LIN {X 0,Y 571.176,Z 836.782,A -85,B 0,C 180,E1 -9234.219,E2 -9234.219} C_VEL
LIN {X 0,Y 568.338,Z 859.351,A -85,B 0,C 180,E1 -9235.423,E2 -9235.423} C_VEL
LIN {X 0,Y 565.653,Z 878.944,A -85,B 0,C 180,E1 -9236.651,E2 -9236.651} C_VEL
LIN {X 0,Y 562.465,Z 900.787,A -85,B 0,C 180,E1 -9238.251,E2 -9238.251} C_VEL
LIN {X 0,Y 559.839,Z 917.889,A -85,B 0,C 180,E1 -9239.698,E2 -9239.698} C_VEL
LIN {X 0,Y 556.887,Z 936.762,A -85,B 0,C 180,E1 -9241.522,E2 -9241.522} C_VEL
LIN {X 0,Y 554.378,Z 952.803,A -85,B 0,C 180,E1 -9243.314,E2 -9243.314} C_VEL
LIN {X 0,Y 551.914,Z 969.075,A -85,B 0,C 180,E1 -9245.375,E2 -9245.375} C_VEL
LIN {X 0,Y 549.794,Z 983.496,A -85,B 0,C 180,E1 -9247.501,E2 -9247.501} C_VEL
LIN {X 0,Y 548.027,Z 996.716,A -85,B 0,C 180,E1 -9249.717,E2 -9249.717} C_VEL
LIN {X 0,Y 546.569,Z 1008.744,A -85,B 0,C 180,E1 -9252.101,E2 -9252.101} C_VEL
LIN {X 0,Y 545.53,Z 1019.1,A -85,B 0,C 180,E1 -9254.479,E2 -9254.479} C_VEL
LIN {X 0,Y 544.771,Z 1027.944,A -85,B 0,C 180,E1 -9256.953,E2 -9256.953} C_VEL
LIN {X 0,Y 544.345,Z 1034.638,A -85,B 0,C 180,E1 -9259.201,E2 -9259.201} C_VEL
LIN {X 0,Y 544.06,Z 1040.823,A -85,B 0,C 180,E1 -9261.865,E2 -9261.865} C_VEL
LIN {X 0,Y 543.971,Z 1044.474,A -85,B 0,C 180,E1 -9263.986,E2 -9263.986} C_VEL
LIN {X 0,Y 543.924,Z 1047.387,A -85,B 0,C 180,E1 -9266.417,E2 -9266.417} C_VEL
LIN {X 0,Y 543.915,Z 1048.764,A -85,B 0,C 180,E1 -9268.947,E2 -9268.947} C_VEL
LIN {X 0,Y 543.919,Z 1048.761,A -85,B 0,C 180,E1 -9271.159,E2 -9271.159} C_VEL
LIN {X 0,Y 543.927,Z 1047.259,A -85,B 0,C 180,E1 -9273.795,E2 -9273.795} C_VEL
LIN {X 0,Y 543.971,Z 1044.452,A -85,B 0,C 180,E1 -9276.12,E2 -9276.12} C_VEL
LIN {X 0,Y 544.08,Z 1040.589,A -85,B 0,C 180,E1 -9278.348,E2 -9278.348} C_VEL
LIN {X 0,Y 544.362,Z 1034.293,A -85,B 0,C 180,E1 -9281.013,E2 -9281.013} C_VEL
LIN {X 0,Y 544.777,Z 1027.888,A -85,B 0,C 180,E1 -9283.155,E2 -9283.155} C_VEL
LIN {X 0,Y 545.538,Z 1019.019,A -85,B 0,C 180,E1 -9285.63,E2 -9285.63} C_VEL
LIN {X 0,Y 546.583,Z 1008.645,A -85,B 0,C 180,E1 -9288.009,E2 -9288.009} C_VEL
LIN {X 0,Y 548.043,Z 996.594,A -85,B 0,C 180,E1 -9290.394,E2 -9290.394} C_VEL
LIN {X 0,Y 549.866,Z 982.95,A -85,B 0,C 180,E1 -9292.675,E2 -9292.675} C_VEL
LIN {X 0,Y 552.067,Z 968.089,A -85,B 0,C 180,E1 -9294.851,E2 -9294.851} C_VEL
LIN {X 0,Y 554.409,Z 952.604,A -85,B 0,C 180,E1 -9296.8,E2 -9296.8} C_VEL
LIN {X 0,Y 557.001,Z 936.1,A -85,B 0,C 180,E1 -9298.64,E2 -9298.64} C_VEL
LIN {X 0,Y 559.829,Z 918.013,A -85,B 0,C 180,E1 -9300.382,E2 -9300.382} C_VEL
LIN {X 0,Y 562.409,Z 901.202,A -85,B 0,C 180,E1 -9301.807,E2 -9301.807} C_VEL
LIN {X 0,Y 565.502,Z 880.175,A -85,B 0,C 180,E1 -9303.36,E2 -9303.36} C_VEL
LIN {X 0,Y 568.145,Z 860.831,A -85,B 0,C 180,E1 -9304.581,E2 -9304.581} C_VEL
LIN {X 0,Y 570.995,Z 838.465,A -85,B 0,C 180,E1 -9305.795,E2 -9305.795} C_VEL
LIN {X 0,Y 573.356,Z 817.368,A -85,B 0,C 180,E1 -9306.739,E2 -9306.739} C_VEL
LIN {X 0,Y 575.397,Z 796.537,A -85,B 0,C 180,E1 -9307.523,E2 -9307.523} C_VEL
LIN {X 0,Y 577.39,Z 771.878,A -85,B 0,C 180,E1 -9308.254,E2 -9308.254} C_VEL
LIN {X 0,Y 578.666,Z 751.524,A -85,B 0,C 180,E1 -9308.716,E2 -9308.716} C_VEL
LIN {X 0,Y 579.729,Z 725.617,A -85,B 0,C 180,E1 -9309.143,E2 -9309.143} C_VEL
LIN {X 0,Y 586.415,Z 471.71,A -85,B 0,C 180,E1 -9312.634,E2 -9312.634} C_VEL
LIN {X 0,Y 587.803,Z 417.401,A -85,B 0,C 180,E1 -9313.399,E2 -9313.399} C_VEL
LIN {X 0,Y 574.092,Z 395,A -85,B 0,C 180,E1 -9315.104,E2 -9315.104} C_VEL
LIN {X 0,Y 562.129,Z 377.006,A -85,B 0,C 180,E1 -9316.677,E2 -9316.677} C_VEL
LIN {X 0,Y 555.49,Z 368.058,A -85,B 0,C 180,E1 -9317.58,E2 -9317.58} C_VEL
LIN {X 0,Y 552.526,Z 363.838,A -85,B 0,C 180,E1 -9318,E2 -9318} C_VEL
LIN {X 0,Y 549.725,Z 359.959,A -85,B 0,C 180,E1 -9318.402,E2 -9318.402} C_VEL
LIN {X 0,Y 548.841,Z 358.788,A -85,B 0,C 180,E1 -9318.529,E2 -9318.529} C_VEL
LIN {X 0,Y 546.385,Z 356.008,A -85,B 0,C 180,E1 -9318.878,E2 -9318.878} C_VEL
LIN {X 0,Y 545.511,Z 353.224,A -85,B 0,C 180,E1 -9319.041,E2 -9319.041} C_VEL
LIN {X 0,Y 545.509,Z 353.268,A -85,B 0,C 180,E1 -9322.383,E2 -9322.383} C_VEL
LIN {X 0,Y 545.559,Z 353.26,A -85,B 0,C 180,E1 -9325.632,E2 -9325.632} C_VEL
LIN {X 0,Y 545.501,Z 353.265,A -85,B 0,C 180,E1 -9328.875,E2 -9328.875} C_VEL
LIN {X 0,Y 545.543,Z 353.258,A -85,B 0,C 180,E1 -9332.136,E2 -9332.136} C_VEL
LIN {X 0,Y 545.515,Z 353.271,A -85,B 0,C 180,E1 -9335.297,E2 -9335.297} C_VEL
LIN {X 0,Y 545.507,Z 353.277,A -85,B 0,C 180,E1 -9338.72,E2 -9338.72} C_VEL
LIN {X 0,Y 545.562,Z 353.271,A -85,B 0,C 180,E1 -9341.956,E2 -9341.956} C_VEL
LIN {X 0,Y 545.5,Z 353.262,A -85,B 0,C 180,E1 -9345.239,E2 -9345.239} C_VEL
LIN {X 0,Y 545.524,Z 353.257,A -85,B 0,C 180,E1 -9348.583,E2 -9348.583} C_VEL
LIN {X 0,Y 545.533,Z 353.279,A -85,B 0,C 180,E1 -9351.79,E2 -9351.79} C_VEL
LIN {X 0,Y 545.502,Z 353.273,A -85,B 0,C 180,E1 -9355.058,E2 -9355.058} C_VEL
LIN {X 0,Y 545.562,Z 353.252,A -85,B 0,C 180,E1 -9358.32,E2 -9358.32} C_VEL
LIN {X 0,Y 545.501,Z 353.279,A -85,B 0,C 180,E1 -9361.47,E2 -9361.47} C_VEL
LIN {X 0,Y 545.528,Z 353.276,A -85,B 0,C 180,E1 -9364.837,E2 -9364.837} C_VEL
LIN {X 0,Y 545.525,Z 353.257,A -85,B 0,C 180,E1 -9368.007,E2 -9368.007} C_VEL
LIN {X 0,Y 545.503,Z 353.271,A -85,B 0,C 180,E1 -9371.311,E2 -9371.311} C_VEL
LIN {X 0,Y 545.571,Z 353.272,A -85,B 0,C 180,E1 -9374.605,E2 -9374.605} C_VEL
LIN {X 0,Y 545.503,Z 353.27,A -85,B 0,C 180,E1 -9377.825,E2 -9377.825} C_VEL
LIN {X 0,Y 545.522,Z 353.261,A -85,B 0,C 180,E1 -9381.167,E2 -9381.167} C_VEL
LIN {X 0,Y 545.522,Z 353.262,A -85,B 0,C 180,E1 -9384.241,E2 -9384.241} C_VEL
LIN {X 0,Y 545.503,Z 353.267,A -85,B 0,C 180,E1 -9387.629,E2 -9387.629} C_VEL
LIN {X 0,Y 545.571,Z 353.262,A -85,B 0,C 180,E1 -9390.753,E2 -9390.753} C_VEL
LIN {X 0,Y 545.502,Z 353.27,A -85,B 0,C 180,E1 -9394.055,E2 -9394.055} C_VEL
LIN {X 0,Y 545.53,Z 353.267,A -85,B 0,C 180,E1 -9397.35,E2 -9397.35} C_VEL
LIN {X 0,Y 545.578,Z 353.397,A -85,B 0,C 180,E1 -9398.84,E2 -9398.84} C_VEL
LIN {X 0,Y 546.798,Z 356.681,A -85,B 0,C 180,E1 -9399.386,E2 -9399.386} C_VEL
LIN {X 0,Y 552.392,Z 369.121,A -85,B 0,C 180,E1 -9401.491,E2 -9401.491} C_VEL
LIN {X 0,Y 553.905,Z 372.53,A -85,B 0,C 180,E1 -9401.993,E2 -9401.993} C_VEL
LIN {X 0,Y 567.117,Z 392.673,A -85,B 0,C 180,E1 -9403.808,E2 -9403.808} C_VEL
LIN {X 0,Y 577.736,Z 409.877,A -85,B 0,C 180,E1 -9405.184,E2 -9405.184} C_VEL
LIN {X 0,Y 587.88,Z 427.42,A -85,B 0,C 180,E1 -9406.442,E2 -9406.442} C_VEL
LIN {X 0,Y 580.977,Z 687.347,A -85,B 0,C 180,E1 -9410.026,E2 -9410.026} C_VEL
LIN {X 0,Y 578.837,Z 765.694,A -85,B 0,C 180,E1 -9411.119,E2 -9411.119} C_VEL
LIN {X 0,Y 577.261,Z 791.324,A -85,B 0,C 180,E1 -9411.637,E2 -9411.637} C_VEL
LIN {X 0,Y 575.512,Z 813.307,A -85,B 0,C 180,E1 -9412.236,E2 -9412.236} C_VEL
LIN {X 0,Y 573.112,Z 838.377,A -85,B 0,C 180,E1 -9413.118,E2 -9413.118} C_VEL
LIN {X 0,Y 570.954,Z 857.811,A -85,B 0,C 180,E1 -9413.955,E2 -9413.955} C_VEL
LIN {X 0,Y 568.235,Z 880.101,A -85,B 0,C 180,E1 -9415.085,E2 -9415.085} C_VEL
LIN {X 0,Y 565.429,Z 900.717,A -85,B 0,C 180,E1 -9416.334,E2 -9416.334} C_VEL
LIN {X 0,Y 562.638,Z 920.354,A -85,B 0,C 180,E1 -9417.699,E2 -9417.699} C_VEL
LIN {X 0,Y 559.633,Z 940.46,A -85,B 0,C 180,E1 -9419.329,E2 -9419.329} C_VEL
LIN {X 0,Y 557.091,Z 957.393,A -85,B 0,C 180,E1 -9420.896,E2 -9420.896} C_VEL
LIN {X 0,Y 554.163,Z 976.778,A -85,B 0,C 180,E1 -9422.955,E2 -9422.955} C_VEL
LIN {X 0,Y 551.957,Z 991.957,A -85,B 0,C 180,E1 -9424.804,E2 -9424.804} C_VEL
LIN {X 0,Y 549.688,Z 1008.329,A -85,B 0,C 180,E1 -9427.091,E2 -9427.091} C_VEL
LIN {X 0,Y 548.053,Z 1021.183,A -85,B 0,C 180,E1 -9429.16,E2 -9429.16} C_VEL
LIN {X 0,Y 546.495,Z 1034.957,A -85,B 0,C 180,E1 -9431.73,E2 -9431.73} C_VEL
LIN {X 0,Y 545.565,Z 1044.545,A -85,B 0,C 180,E1 -9433.824,E2 -9433.824} C_VEL
LIN {X 0,Y 544.805,Z 1054.264,A -85,B 0,C 180,E1 -9436.305,E2 -9436.305} C_VEL
LIN {X 0,Y 544.339,Z 1061.766,A -85,B 0,C 180,E1 -9438.665,E2 -9438.665} C_VEL
LIN {X 0,Y 544.07,Z 1067.86,A -85,B 0,C 180,E1 -9441.013,E2 -9441.013} C_VEL
LIN {X 0,Y 543.949,Z 1072.768,A -85,B 0,C 180,E1 -9443.562,E2 -9443.562} C_VEL
LIN {X 0,Y 543.918,Z 1075.605,A -85,B 0,C 180,E1 -9445.677,E2 -9445.677} C_VEL
LIN {X 0,Y 543.91,Z 1077.486,A -85,B 0,C 180,E1 -9447.998,E2 -9447.998} C_VEL
LIN {X 0,Y 543.902,Z 1077.918,A -85,B 0,C 180,E1 -9450.527,E2 -9450.527} C_VEL
LIN {X 0,Y 543.912,Z 1077.002,A -85,B 0,C 180,E1 -9452.739,E2 -9452.739} C_VEL
LIN {X 0,Y 543.933,Z 1074.678,A -85,B 0,C 180,E1 -9455.168,E2 -9455.168} C_VEL
LIN {X 0,Y 543.986,Z 1070.708,A -85,B 0,C 180,E1 -9457.605,E2 -9457.605} C_VEL
LIN {X 0,Y 544.145,Z 1066.052,A -85,B 0,C 180,E1 -9459.733,E2 -9459.733} C_VEL
LIN {X 0,Y 544.483,Z 1059.283,A -85,B 0,C 180,E1 -9462.192,E2 -9462.192} C_VEL
LIN {X 0,Y 545.03,Z 1051.049,A -85,B 0,C 180,E1 -9464.556,E2 -9464.556} C_VEL
LIN {X 0,Y 545.787,Z 1042.224,A -85,B 0,C 180,E1 -9466.716,E2 -9466.716} C_VEL
LIN {X 0,Y 547.006,Z 1030.198,A -85,B 0,C 180,E1 -9469.21,E2 -9469.21} C_VEL
LIN {X 0,Y 548.367,Z 1018.538,A -85,B 0,C 180,E1 -9471.289,E2 -9471.289} C_VEL
LIN {X 0,Y 550.294,Z 1003.933,A -85,B 0,C 180,E1 -9473.562,E2 -9473.562} C_VEL
LIN {X 0,Y 552.314,Z 989.393,A -85,B 0,C 180,E1 -9475.522,E2 -9475.522} C_VEL
LIN {X 0,Y 554.856,Z 972.384,A -85,B 0,C 180,E1 -9477.548,E2 -9477.548} C_VEL
LIN {X 0,Y 557.435,Z 954.991,A -85,B 0,C 180,E1 -9479.336,E2 -9479.336} C_VEL
LIN {X 0,Y 560.299,Z 936.15,A -85,B 0,C 180,E1 -9481.047,E2 -9481.047} C_VEL
LIN {X 0,Y 563.178,Z 916.498,A -85,B 0,C 180,E1 -9482.578,E2 -9482.578} C_VEL
LIN {X 0,Y 565.814,Z 897.977,A -85,B 0,C 180,E1 -9483.842,E2 -9483.842} C_VEL
LIN {X 0,Y 568.871,Z 874.652,A -85,B 0,C 180,E1 -9485.206,E2 -9485.206} C_VEL
LIN {X 0,Y 571.297,Z 854.713,A -85,B 0,C 180,E1 -9486.187,E2 -9486.187} C_VEL
LIN {X 0,Y 573.858,Z 830.892,A -85,B 0,C 180,E1 -9487.17,E2 -9487.17} C_VEL
LIN {X 0,Y 575.888,Z 808.712,A -85,B 0,C 180,E1 -9487.898,E2 -9487.898} C_VEL
LIN {X 0,Y 577.792,Z 784.379,A -85,B 0,C 180,E1 -9488.523,E2 -9488.523} C_VEL
LIN {X 0,Y 579.016,Z 760.564,A -85,B 0,C 180,E1 -9488.957,E2 -9488.957} C_VEL
LIN {X 0,Y 585.161,Z 525.146,A -85,B 0,C 180,E1 -9492.202,E2 -9492.202} C_VEL
LIN {X 0,Y 587.734,Z 427.102,A -85,B 0,C 180,E1 -9493.57,E2 -9493.57} C_VEL
LIN {X 0,Y 574.449,Z 404.387,A -85,B 0,C 180,E1 -9495.227,E2 -9495.227} C_VEL
LIN {X 0,Y 561.317,Z 383.659,A -85,B 0,C 180,E1 -9496.963,E2 -9496.963} C_VEL
LIN {X 0,Y 553.323,Z 371.554,A -85,B 0,C 180,E1 -9498.117,E2 -9498.117} C_VEL
LIN {X 0,Y 548.816,Z 361.059,A -85,B 0,C 180,E1 -9499.838,E2 -9499.838} C_VEL
LIN {X 0,Y 545.6,Z 353.509,A -85,B 0,C 180,E1 -9501.127,E2 -9501.127} C_VEL
LIN {X 0,Y 545.5,Z 353.212,A -85,B 0,C 180,E1 -9504.346,E2 -9504.346} C_VEL
LIN {X 0,Y 545.514,Z 353.271,A -85,B 0,C 180,E1 -9507.765,E2 -9507.765} C_VEL
LIN {X 0,Y 545.536,Z 353.273,A -85,B 0,C 180,E1 -9510.821,E2 -9510.821} C_VEL
LIN {X 0,Y 545.506,Z 353.278,A -85,B 0,C 180,E1 -9514.156,E2 -9514.156} C_VEL
LIN {X 0,Y 545.562,Z 353.271,A -85,B 0,C 180,E1 -9517.477,E2 -9517.477} C_VEL
LIN {X 0,Y 545.513,Z 353.269,A -85,B 0,C 180,E1 -9520.735,E2 -9520.735} C_VEL
LIN {X 0,Y 545.508,Z 353.262,A -85,B 0,C 180,E1 -9524.15,E2 -9524.15} C_VEL
LIN {X 0,Y 545.555,Z 353.263,A -85,B 0,C 180,E1 -9527.295,E2 -9527.295} C_VEL
LIN {X 0,Y 545.504,Z 353.278,A -85,B 0,C 180,E1 -9530.611,E2 -9530.611} C_VEL
LIN {X 0,Y 545.544,Z 353.262,A -85,B 0,C 180,E1 -9533.898,E2 -9533.898} C_VEL
LIN {X 0,Y 545.516,Z 353.259,A -85,B 0,C 180,E1 -9537.058,E2 -9537.058} C_VEL
LIN {X 0,Y 545.511,Z 353.274,A -85,B 0,C 180,E1 -9540.42,E2 -9540.42} C_VEL
LIN {X 0,Y 545.56,Z 353.266,A -85,B 0,C 180,E1 -9543.678,E2 -9543.678} C_VEL
LIN {X 0,Y 545.505,Z 353.257,A -85,B 0,C 180,E1 -9546.948,E2 -9546.948} C_VEL
LIN {X 0,Y 545.537,Z 353.264,A -85,B 0,C 180,E1 -9550.241,E2 -9550.241} C_VEL
LIN {X 0,Y 545.529,Z 353.275,A -85,B 0,C 180,E1 -9553.461,E2 -9553.461} C_VEL
LIN {X 0,Y 545.51,Z 353.27,A -85,B 0,C 180,E1 -9556.834,E2 -9556.834} C_VEL
LIN {X 0,Y 545.566,Z 353.255,A -85,B 0,C 180,E1 -9560.043,E2 -9560.043} C_VEL
LIN {X 0,Y 545.508,Z 353.271,A -85,B 0,C 180,E1 -9563.209,E2 -9563.209} C_VEL
LIN {X 0,Y 545.537,Z 353.272,A -85,B 0,C 180,E1 -9566.565,E2 -9566.565} C_VEL
LIN {X 0,Y 545.528,Z 353.277,A -85,B 0,C 180,E1 -9569.682,E2 -9569.682} C_VEL
LIN {X 0,Y 545.512,Z 353.278,A -85,B 0,C 180,E1 -9573.108,E2 -9573.108} C_VEL
LIN {X 0,Y 545.563,Z 353.271,A -85,B 0,C 180,E1 -9576.43,E2 -9576.43} C_VEL
LIN {X 0,Y 545.515,Z 353.273,A -85,B 0,C 180,E1 -9579.662,E2 -9579.662} C_VEL
LIN {X 0,Y 545.546,Z 353.48,A -85,B 0,C 180,E1 -9581.076,E2 -9581.076} C_VEL
LIN {X 0,Y 546.721,Z 356.617,A -85,B 0,C 180,E1 -9581.279,E2 -9581.279} C_VEL
LIN {X 0,Y 549.657,Z 359.833,A -85,B 0,C 180,E1 -9581.691,E2 -9581.691} C_VEL
LIN {X 0,Y 552.394,Z 363.737,A -85,B 0,C 180,E1 -9582.086,E2 -9582.086} C_VEL
LIN {X 0,Y 554.158,Z 366.201,A -85,B 0,C 180,E1 -9582.336,E2 -9582.336} C_VEL
LIN {X 0,Y 563.303,Z 378.672,A -85,B 0,C 180,E1 -9583.582,E2 -9583.582} C_VEL
LIN {X 0,Y 577.707,Z 400.638,A -85,B 0,C 180,E1 -9585.452,E2 -9585.452} C_VEL
LIN {X 0,Y 587.857,Z 417.84,A -85,B 0,C 180,E1 -9586.709,E2 -9586.709} C_VEL
LIN {X 0,Y 581.199,Z 666.938,A -85,B 0,C 180,E1 -9590.147,E2 -9590.147} C_VEL
LIN {X 0,Y 579.851,Z 720.042,A -85,B 0,C 180,E1 -9590.873,E2 -9590.873} C_VEL
LIN {X 0,Y 578.841,Z 727.729,A -85,B 0,C 180,E1 -9590.911,E2 -9590.911} C_VEL
LIN {X 0,Y 573.414,Z 747.093,A -85,B 0,C 180,E1 -9590.84,E2 -9590.84} C_VEL
LIN {X 0,Y 572.239,Z 754.709,A -85,B 0,C 180,E1 -9590.936,E2 -9590.936} C_VEL
LIN {X 0,Y 570.608,Z 778.562,A -85,B 0,C 180,E1 -9591.508,E2 -9591.508} C_VEL
LIN {X 0,Y 568.556,Z 801.206,A -85,B 0,C 180,E1 -9592.233,E2 -9592.233} C_VEL
LIN {X 0,Y 566.233,Z 823.809,A -85,B 0,C 180,E1 -9593.124,E2 -9593.124} C_VEL
LIN {X 0,Y 563.444,Z 846.211,A -85,B 0,C 180,E1 -9594.21,E2 -9594.21} C_VEL
LIN {X 0,Y 560.814,Z 865.965,A -85,B 0,C 180,E1 -9595.337,E2 -9595.337} C_VEL
LIN {X 0,Y 557.629,Z 887.571,A -85,B 0,C 180,E1 -9596.784,E2 -9596.784} C_VEL
LIN {X 0,Y 554.905,Z 904.986,A -85,B 0,C 180,E1 -9598.132,E2 -9598.132} C_VEL
LIN {X 0,Y 551.74,Z 924.582,A -85,B 0,C 180,E1 -9599.868,E2 -9599.868} C_VEL
LIN {X 0,Y 548.917,Z 941.636,A -85,B 0,C 180,E1 -9601.621,E2 -9601.621} C_VEL
LIN {X 0,Y 546.187,Z 958.486,A -85,B 0,C 180,E1 -9603.586,E2 -9603.586} C_VEL
LIN {X 0,Y 543.711,Z 973.867,A -85,B 0,C 180,E1 -9605.673,E2 -9605.673} C_VEL
LIN {X 0,Y 541.581,Z 988.153,A -85,B 0,C 180,E1 -9607.875,E2 -9607.875} C_VEL
LIN {X 0,Y 539.759,Z 1001.146,A -85,B 0,C 180,E1 -9610.231,E2 -9610.231} C_VEL
LIN {X 0,Y 538.386,Z 1012.519,A -85,B 0,C 180,E1 -9612.602,E2 -9612.602} C_VEL
LIN {X 0,Y 537.371,Z 1022.142,A -85,B 0,C 180,E1 -9615.011,E2 -9615.011} C_VEL
LIN {X 0,Y 536.721,Z 1029.902,A -85,B 0,C 180,E1 -9617.301,E2 -9617.301} C_VEL
LIN {X 0,Y 536.241,Z 1037.284,A -85,B 0,C 180,E1 -9620.014,E2 -9620.014} C_VEL
LIN {X 0,Y 536.039,Z 1041.852,A -85,B 0,C 180,E1 -9622.174,E2 -9622.174} C_VEL
LIN {X 0,Y 535.95,Z 1045.789,A -85,B 0,C 180,E1 -9624.648,E2 -9624.648} C_VEL
LIN {X 0,Y 535.912,Z 1048.186,A -85,B 0,C 180,E1 -9627.22,E2 -9627.22} C_VEL
LIN {X 0,Y 535.905,Z 1049.089,A -85,B 0,C 180,E1 -9629.466,E2 -9629.466} C_VEL
LIN {X 0,Y 535.922,Z 1048.644,A -85,B 0,C 180,E1 -9632.139,E2 -9632.139} C_VEL
LIN {X 0,Y 535.939,Z 1046.802,A -85,B 0,C 180,E1 -9634.494,E2 -9634.494} C_VEL
LIN {X 0,Y 536.005,Z 1043.568,A -85,B 0,C 180,E1 -9636.965,E2 -9636.965} C_VEL
LIN {X 0,Y 536.199,Z 1038.491,A -85,B 0,C 180,E1 -9639.553,E2 -9639.553} C_VEL
LIN {X 0,Y 536.52,Z 1032.719,A -85,B 0,C 180,E1 -9641.83,E2 -9641.83} C_VEL
LIN {X 0,Y 537.196,Z 1024.041,A -85,B 0,C 180,E1 -9644.559,E2 -9644.559} C_VEL
LIN {X 0,Y 538.025,Z 1015.615,A -85,B 0,C 180,E1 -9646.742,E2 -9646.742} C_VEL
LIN {X 0,Y 539.307,Z 1004.753,A -85,B 0,C 180,E1 -9649.157,E2 -9649.157} C_VEL
LIN {X 0,Y 540.939,Z 992.42,A -85,B 0,C 180,E1 -9651.469,E2 -9651.469} C_VEL
LIN {X 0,Y 542.95,Z 979.012,A -85,B 0,C 180,E1 -9653.67,E2 -9653.67} C_VEL
LIN {X 0,Y 545.284,Z 963.895,A -85,B 0,C 180,E1 -9655.795,E2 -9655.795} C_VEL
LIN {X 0,Y 547.857,Z 948.236,A -85,B 0,C 180,E1 -9657.736,E2 -9657.736} C_VEL
LIN {X 0,Y 550.788,Z 930.376,A -85,B 0,C 180,E1 -9659.65,E2 -9659.65} C_VEL
LIN {X 0,Y 553.53,Z 913.605,A -85,B 0,C 180,E1 -9661.227,E2 -9661.227} C_VEL
LIN {X 0,Y 556.897,Z 892.328,A -85,B 0,C 180,E1 -9662.958,E2 -9662.958} C_VEL
LIN {X 0,Y 559.672,Z 873.934,A -85,B 0,C 180,E1 -9664.247,E2 -9664.247} C_VEL
LIN {X 0,Y 562.89,Z 850.792,A -85,B 0,C 180,E1 -9665.637,E2 -9665.637} C_VEL
LIN {X 0,Y 565.275,Z 831.922,A -85,B 0,C 180,E1 -9666.592,E2 -9666.592} C_VEL
LIN {X 0,Y 567.85,Z 809.167,A -85,B 0,C 180,E1 -9667.571,E2 -9667.571} C_VEL
LIN {X 0,Y 570.011,Z 785.467,A -85,B 0,C 180,E1 -9668.378,E2 -9668.378} C_VEL
LIN {X 0,Y 571.862,Z 761.537,A -85,B 0,C 180,E1 -9669.018,E2 -9669.018} C_VEL
LIN {X 0,Y 573.127,Z 737.079,A -85,B 0,C 180,E1 -9669.478,E2 -9669.478} C_VEL
LIN {X 0,Y 579.836,Z 496.377,A -85,B 0,C 180,E1 -9672.829,E2 -9672.829} C_VEL
LIN {X 0,Y 581.858,Z 420.664,A -85,B 0,C 180,E1 -9673.904,E2 -9673.904} C_VEL
LIN {X 0,Y 569.342,Z 400.206,A -85,B 0,C 180,E1 -9675.496,E2 -9675.496} C_VEL
LIN {X 0,Y 557.802,Z 382.694,A -85,B 0,C 180,E1 -9677.047,E2 -9677.047} C_VEL
LIN {X 0,Y 548.177,Z 369.608,A -85,B 0,C 180,E1 -9678.398,E2 -9678.398} C_VEL
LIN {X 0,Y 544.811,Z 365.055,A -85,B 0,C 180,E1 -9678.891,E2 -9678.891} C_VEL
LIN {X 0,Y 541.972,Z 361.25,A -85,B 0,C 180,E1 -9679.314,E2 -9679.314} C_VEL
LIN {X 0,Y 541.06,Z 359.842,A -85,B 0,C 180,E1 -9679.455,E2 -9679.455} C_VEL
LIN {X 0,Y 538.501,Z 357.011,A -85,B 0,C 180,E1 -9679.834,E2 -9679.834} C_VEL
LIN {X 0,Y 537.591,Z 354.226,A -85,B 0,C 180,E1 -9680.023,E2 -9680.023} C_VEL
LIN {X 0,Y 537.578,Z 354.255,A -85,B 0,C 180,E1 -9683.111,E2 -9683.111} C_VEL
LIN {X 0,Y 537.571,Z 354.26,A -85,B 0,C 180,E1 -9686.466,E2 -9686.466} C_VEL
LIN {X 0,Y 537.629,Z 354.25,A -85,B 0,C 180,E1 -9689.734,E2 -9689.734} C_VEL
LIN {X 0,Y 537.565,Z 354.252,A -85,B 0,C 180,E1 -9693.009,E2 -9693.009} C_VEL
LIN {X 0,Y 537.583,Z 354.248,A -85,B 0,C 180,E1 -9696.428,E2 -9696.428} C_VEL
LIN {X 0,Y 537.587,Z 354.253,A -85,B 0,C 180,E1 -9699.533,E2 -9699.533} C_VEL
LIN {X 0,Y 537.564,Z 354.267,A -85,B 0,C 180,E1 -9702.909,E2 -9702.909} C_VEL
LIN {X 0,Y 537.621,Z 354.26,A -85,B 0,C 180,E1 -9706.228,E2 -9706.228} C_VEL
LIN {X 0,Y 537.57,Z 354.245,A -85,B 0,C 180,E1 -9709.497,E2 -9709.497} C_VEL
LIN {X 0,Y 537.567,Z 354.254,A -85,B 0,C 180,E1 -9712.948,E2 -9712.948} C_VEL
LIN {X 0,Y 537.622,Z 354.263,A -85,B 0,C 180,E1 -9716.268,E2 -9716.268} C_VEL
LIN {X 0,Y 537.567,Z 354.256,A -85,B 0,C 180,E1 -9719.574,E2 -9719.574} C_VEL
LIN {X 0,Y 537.571,Z 354.242,A -85,B 0,C 180,E1 -9722.985,E2 -9722.985} C_VEL
LIN {X 0,Y 537.619,Z 354.255,A -85,B 0,C 180,E1 -9726.3,E2 -9726.3} C_VEL
LIN {X 0,Y 537.562,Z 354.266,A -85,B 0,C 180,E1 -9729.529,E2 -9729.529} C_VEL
LIN {X 0,Y 537.594,Z 354.249,A -85,B 0,C 180,E1 -9732.897,E2 -9732.897} C_VEL
LIN {X 0,Y 537.575,Z 354.252,A -85,B 0,C 180,E1 -9735.979,E2 -9735.979} C_VEL
LIN {X 0,Y 537.565,Z 354.263,A -85,B 0,C 180,E1 -9739.448,E2 -9739.448} C_VEL
LIN {X 0,Y 537.631,Z 354.26,A -85,B 0,C 180,E1 -9742.758,E2 -9742.758} C_VEL
LIN {X 0,Y 537.571,Z 354.266,A -85,B 0,C 180,E1 -9746.053,E2 -9746.053} C_VEL
LIN {X 0,Y 537.572,Z 354.269,A -85,B 0,C 180,E1 -9749.532,E2 -9749.532} C_VEL
LIN {X 0,Y 537.621,Z 354.266,A -85,B 0,C 180,E1 -9752.791,E2 -9752.791} C_VEL
LIN {X 0,Y 537.563,Z 354.271,A -85,B 0,C 180,E1 -9755.999,E2 -9755.999} C_VEL
LIN {X 0,Y 537.588,Z 354.456,A -85,B 0,C 180,E1 -9757.943,E2 -9757.943} C_VEL
LIN {X 0,Y 539.011,Z 357.914,A -85,B 0,C 180,E1 -9758.557,E2 -9758.557} C_VEL
LIN {X 0,Y 544.971,Z 371.337,A -85,B 0,C 180,E1 -9760.894,E2 -9760.894} C_VEL
LIN {X 0,Y 558.146,Z 391.043,A -85,B 0,C 180,E1 -9762.815,E2 -9762.815} C_VEL
LIN {X 0,Y 572.183,Z 413.656,A -85,B 0,C 180,E1 -9764.698,E2 -9764.698} C_VEL
LIN {X 0,Y 581.977,Z 430.756,A -85,B 0,C 180,E1 -9765.946,E2 -9765.946} C_VEL
LIN {X 0,Y 574.793,Z 689.065,A -85,B 0,C 180,E1 -9769.538,E2 -9769.538} C_VEL
LIN {X 0,Y 572.602,Z 765.604,A -85,B 0,C 180,E1 -9770.617,E2 -9770.617} C_VEL
LIN {X 0,Y 570.971,Z 791.119,A -85,B 0,C 180,E1 -9771.135,E2 -9771.135} C_VEL
LIN {X 0,Y 569.152,Z 813.036,A -85,B 0,C 180,E1 -9771.736,E2 -9771.736} C_VEL
LIN {X 0,Y 566.64,Z 838.166,A -85,B 0,C 180,E1 -9772.626,E2 -9772.626} C_VEL
LIN {X 0,Y 564.26,Z 858.743,A -85,B 0,C 180,E1 -9773.522,E2 -9773.522} C_VEL
LIN {X 0,Y 561.219,Z 882.193,A -85,B 0,C 180,E1 -9774.742,E2 -9774.742} C_VEL
LIN {X 0,Y 558.509,Z 901.289,A -85,B 0,C 180,E1 -9775.919,E2 -9775.919} C_VEL
LIN {X 0,Y 555.448,Z 921.881,A -85,B 0,C 180,E1 -9777.375,E2 -9777.375} C_VEL
LIN {X 0,Y 552.325,Z 941.616,A -85,B 0,C 180,E1 -9779.014,E2 -9779.014} C_VEL
LIN {X 0,Y 549.374,Z 960.531,A -85,B 0,C 180,E1 -9780.806,E2 -9780.806} C_VEL
LIN {X 0,Y 546.493,Z 978.429,A -85,B 0,C 180,E1 -9782.78,E2 -9782.78} C_VEL
LIN {X 0,Y 543.976,Z 995.138,A -85,B 0,C 180,E1 -9784.874,E2 -9784.874} C_VEL
LIN {X 0,Y 541.756,Z 1010.235,A -85,B 0,C 180,E1 -9787.081,E2 -9787.081} C_VEL
LIN {X 0,Y 540.009,Z 1023.534,A -85,B 0,C 180,E1 -9789.289,E2 -9789.289} C_VEL
LIN {X 0,Y 538.53,Z 1035.959,A -85,B 0,C 180,E1 -9791.713,E2 -9791.713} C_VEL
LIN {X 0,Y 537.51,Z 1046.188,A -85,B 0,C 180,E1 -9794.019,E2 -9794.019} C_VEL
LIN {X 0,Y 536.754,Z 1055.481,A -85,B 0,C 180,E1 -9796.535,E2 -9796.535} C_VEL
LIN {X 0,Y 536.334,Z 1062.164,A -85,B 0,C 180,E1 -9798.711,E2 -9798.711} C_VEL
LIN {X 0,Y 536.054,Z 1068.601,A -85,B 0,C 180,E1 -9801.31,E2 -9801.31} C_VEL
LIN {X 0,Y 535.95,Z 1072.879,A -85,B 0,C 180,E1 -9803.68,E2 -9803.68} C_VEL
LIN {X 0,Y 535.917,Z 1075.622,A -85,B 0,C 180,E1 -9805.827,E2 -9805.827} C_VEL
LIN {X 0,Y 535.901,Z 1077.473,A -85,B 0,C 180,E1 -9808.396,E2 -9808.396} C_VEL
LIN {X 0,Y 535.908,Z 1077.659,A -85,B 0,C 180,E1 -9810.748,E2 -9810.748} C_VEL
LIN {X 0,Y 535.92,Z 1076.65,A -85,B 0,C 180,E1 -9812.994,E2 -9812.994} C_VEL
LIN {X 0,Y 535.941,Z 1073.853,A -85,B 0,C 180,E1 -9815.675,E2 -9815.675} C_VEL
LIN {X 0,Y 536.004,Z 1070.073,A -85,B 0,C 180,E1 -9817.935,E2 -9817.935} C_VEL
LIN {X 0,Y 536.186,Z 1065.059,A -85,B 0,C 180,E1 -9820.204,E2 -9820.204} C_VEL
LIN {X 0,Y 536.601,Z 1057.632,A -85,B 0,C 180,E1 -9822.811,E2 -9822.811} C_VEL
LIN {X 0,Y 537.167,Z 1050.008,A -85,B 0,C 180,E1 -9824.995,E2 -9824.995} C_VEL
LIN {X 0,Y 538.1,Z 1040.134,A -85,B 0,C 180,E1 -9827.408,E2 -9827.408} C_VEL
LIN {X 0,Y 539.415,Z 1028.234,A -85,B 0,C 180,E1 -9829.829,E2 -9829.829} C_VEL
LIN {X 0,Y 541.11,Z 1015.178,A -85,B 0,C 180,E1 -9832.145,E2 -9832.145} C_VEL
LIN {X 0,Y 543.131,Z 1000.593,A -85,B 0,C 180,E1 -9834.354,E2 -9834.354} C_VEL
LIN {X 0,Y 545.523,Z 984.899,A -85,B 0,C 180,E1 -9836.448,E2 -9836.448} C_VEL
LIN {X 0,Y 548.227,Z 967.367,A -85,B 0,C 180,E1 -9838.465,E2 -9838.465} C_VEL
LIN {X 0,Y 550.942,Z 950.442,A -85,B 0,C 180,E1 -9840.18,E2 -9840.18} C_VEL
LIN {X 0,Y 554.063,Z 930.605,A -85,B 0,C 180,E1 -9841.922,E2 -9841.922} C_VEL
LIN {X 0,Y 556.71,Z 913.33,A -85,B 0,C 180,E1 -9843.249,E2 -9843.249} C_VEL
LIN {X 0,Y 559.832,Z 892.112,A -85,B 0,C 180,E1 -9844.67,E2 -9844.67} C_VEL
LIN {X 0,Y 562.666,Z 870.924,A -85,B 0,C 180,E1 -9845.871,E2 -9845.871} C_VEL
LIN {X 0,Y 565.527,Z 848.413,A -85,B 0,C 180,E1 -9846.952,E2 -9846.952} C_VEL
LIN {X 0,Y 567.881,Z 826.214,A -85,B 0,C 180,E1 -9847.819,E2 -9847.819} C_VEL
LIN {X 0,Y 569.869,Z 805.148,A -85,B 0,C 180,E1 -9848.493,E2 -9848.493} C_VEL
LIN {X 0,Y 571.772,Z 779.887,A -85,B 0,C 180,E1 -9849.111,E2 -9849.111} C_VEL
LIN {X 0,Y 572.887,Z 757.978,A -85,B 0,C 180,E1 -9849.499,E2 -9849.499} C_VEL
LIN {X 0,Y 579.526,Z 514.708,A -85,B 0,C 180,E1 -9852.878,E2 -9852.878} C_VEL
LIN {X 0,Y 581.836,Z 430.472,A -85,B 0,C 180,E1 -9854.065,E2 -9854.065} C_VEL
LIN {X 0,Y 569.608,Z 409.402,A -85,B 0,C 180,E1 -9855.628,E2 -9855.628} C_VEL
LIN {X 0,Y 556.891,Z 389.22,A -85,B 0,C 180,E1 -9857.346,E2 -9857.346} C_VEL
LIN {X 0,Y 546.257,Z 373.533,A -85,B 0,C 180,E1 -9858.866,E2 -9858.866} C_VEL
LIN {X 0,Y 544.91,Z 371.213,A -85,B 0,C 180,E1 -9859.113,E2 -9859.113} C_VEL
LIN {X 0,Y 539.334,Z 358.315,A -85,B 0,C 180,E1 -9861.334,E2 -9861.334} C_VEL
LIN {X 0,Y 537.809,Z 355.461,A -85,B 0,C 180,E1 -9861.884,E2 -9861.884} C_VEL
LIN {X 0,Y 537.561,Z 354.251,A -85,B 0,C 180,E1 -9862.096,E2 -9862.096} C_VEL
LIN {X 0,Y 537.592,Z 354.207,A -85,B 0,C 180,E1 -9865.439,E2 -9865.439} C_VEL
LIN {X 0,Y 537.578,Z 354.248,A -85,B 0,C 180,E1 -9868.62,E2 -9868.62} C_VEL
LIN {X 0,Y 537.569,Z 354.248,A -85,B 0,C 180,E1 -9871.928,E2 -9871.928} C_VEL
LIN {X 0,Y 537.624,Z 354.248,A -85,B 0,C 180,E1 -9875.262,E2 -9875.262} C_VEL
LIN {X 0,Y 537.567,Z 354.266,A -85,B 0,C 180,E1 -9878.505,E2 -9878.505} C_VEL
LIN {X 0,Y 537.586,Z 354.267,A -85,B 0,C 180,E1 -9881.904,E2 -9881.904} C_VEL
LIN {X 0,Y 537.603,Z 354.255,A -85,B 0,C 180,E1 -9885.128,E2 -9885.128} C_VEL
LIN {X 0,Y 537.564,Z 354.248,A -85,B 0,C 180,E1 -9888.411,E2 -9888.411} C_VEL
LIN {X 0,Y 537.617,Z 354.247,A -85,B 0,C 180,E1 -9891.766,E2 -9891.766} C_VEL
LIN {X 0,Y 537.577,Z 354.266,A -85,B 0,C 180,E1 -9894.985,E2 -9894.985} C_VEL
LIN {X 0,Y 537.573,Z 354.256,A -85,B 0,C 180,E1 -9898.401,E2 -9898.401} C_VEL
LIN {X 0,Y 537.621,Z 354.243,A -85,B 0,C 180,E1 -9901.599,E2 -9901.599} C_VEL
LIN {X 0,Y 537.568,Z 354.266,A -85,B 0,C 180,E1 -9904.908,E2 -9904.908} C_VEL
LIN {X 0,Y 537.59,Z 354.261,A -85,B 0,C 180,E1 -9908.314,E2 -9908.314} C_VEL
LIN {X 0,Y 537.602,Z 354.242,A -85,B 0,C 180,E1 -9911.588,E2 -9911.588} C_VEL
LIN {X 0,Y 537.567,Z 354.257,A -85,B 0,C 180,E1 -9914.873,E2 -9914.873} C_VEL
LIN {X 0,Y 537.618,Z 354.265,A -85,B 0,C 180,E1 -9918.207,E2 -9918.207} C_VEL
LIN {X 0,Y 537.585,Z 354.262,A -85,B 0,C 180,E1 -9921.495,E2 -9921.495} C_VEL
LIN {X 0,Y 537.575,Z 354.256,A -85,B 0,C 180,E1 -9924.857,E2 -9924.857} C_VEL
LIN {X 0,Y 537.634,Z 354.244,A -85,B 0,C 180,E1 -9928.19,E2 -9928.19} C_VEL
LIN {X 0,Y 537.57,Z 354.25,A -85,B 0,C 180,E1 -9931.386,E2 -9931.386} C_VEL
LIN {X 0,Y 537.598,Z 354.25,A -85,B 0,C 180,E1 -9934.706,E2 -9934.706} C_VEL
LIN {X 0,Y 537.602,Z 354.25,A -85,B 0,C 180,E1 -9937.998,E2 -9937.998} C_VEL
LIN {X 0,Y 537.636,Z 354.434,A -85,B 0,C 180,E1 -9940.111,E2 -9940.111} C_VEL
LIN {X 0,Y 538.84,Z 357.584,A -85,B 0,C 180,E1 -9940.328,E2 -9940.328} C_VEL
LIN {X 0,Y 541.702,Z 360.721,A -85,B 0,C 180,E1 -9940.748,E2 -9940.748} C_VEL
LIN {X 0,Y 544.355,Z 364.654,A -85,B 0,C 180,E1 -9941.151,E2 -9941.151} C_VEL
LIN {X 0,Y 546.128,Z 366.8,A -85,B 0,C 180,E1 -9941.407,E2 -9941.407} C_VEL
LIN {X 0,Y 557.965,Z 382.966,A -85,B 0,C 180,E1 -9943.078,E2 -9943.078} C_VEL
LIN {X 0,Y 570.065,Z 401.329,A -85,B 0,C 180,E1 -9944.697,E2 -9944.697} C_VEL
LIN {X 0,Y 581.968,Z 421.15,A -85,B 0,C 180,E1 -9946.212,E2 -9946.212} C_VEL
LIN {X 0,Y 575.013,Z 669.594,A -85,B 0,C 180,E1 -9949.67,E2 -9949.67} C_VEL
LIN {X 0,Y 572.905,Z 742.243,A -85,B 0,C 180,E1 -9950.696,E2 -9950.696} C_VEL
LIN {X 0,Y 572.239,Z 754.709,A -85,B 0,C 180,E1 -9950.936,E2 -9950.936} C_VEL
LIN {X 0,Y 570.655,Z 763.388,A -85,B 0,C 180,E1 -9951.034,E2 -9951.034} C_VEL
LIN {X 0,Y 564.757,Z 781.433,A -85,B 0,C 180,E1 -9951.134,E2 -9951.134} C_VEL
LIN {X 0,Y 563.443,Z 788.88,A -85,B 0,C 180,E1 -9951.308,E2 -9951.308} C_VEL
LIN {X 0,Y 561.007,Z 813.351,A -85,B 0,C 180,E1 -9952.185,E2 -9952.185} C_VEL
LIN {X 0,Y 558.711,Z 832.731,A -85,B 0,C 180,E1 -9953.036,E2 -9953.036} C_VEL
LIN {X 0,Y 555.992,Z 853.528,A -85,B 0,C 180,E1 -9954.107,E2 -9954.107} C_VEL
LIN {X 0,Y 552.765,Z 875.362,A -85,B 0,C 180,E1 -9955.453,E2 -9955.453} C_VEL
LIN {X 0,Y 549.78,Z 894.359,A -85,B 0,C 180,E1 -9956.809,E2 -9956.809} C_VEL
LIN {X 0,Y 546.345,Z 914.947,A -85,B 0,C 180,E1 -9958.523,E2 -9958.523} C_VEL
LIN {X 0,Y 543.445,Z 931.956,A -85,B 0,C 180,E1 -9960.152,E2 -9960.152} C_VEL
LIN {X 0,Y 540.18,Z 950.741,A -85,B 0,C 180,E1 -9962.227,E2 -9962.227} C_VEL
LIN {X 0,Y 537.675,Z 965.397,A -85,B 0,C 180,E1 -9964.086,E2 -9964.086} C_VEL
LIN {X 0,Y 535.036,Z 981.459,A -85,B 0,C 180,E1 -9966.426,E2 -9966.426} C_VEL
LIN {X 0,Y 533.161,Z 993.581,A -85,B 0,C 180,E1 -9968.467,E2 -9968.467} C_VEL
LIN {X 0,Y 531.402,Z 1006.143,A -85,B 0,C 180,E1 -9970.889,E2 -9970.889} C_VEL
LIN {X 0,Y 530.133,Z 1016.378,A -85,B 0,C 180,E1 -9973.227,E2 -9973.227} C_VEL
LIN {X 0,Y 529.197,Z 1025.552,A -85,B 0,C 180,E1 -9975.669,E2 -9975.669} C_VEL
LIN {X 0,Y 528.548,Z 1033.286,A -85,B 0,C 180,E1 -9978.211,E2 -9978.211} C_VEL
LIN {X 0,Y 528.211,Z 1039.001,A -85,B 0,C 180,E1 -9980.521,E2 -9980.521} C_VEL
LIN {X 0,Y 528.005,Z 1044.122,A -85,B 0,C 180,E1 -9983.257,E2 -9983.257} C_VEL
LIN {X 0,Y 527.944,Z 1047.034,A -85,B 0,C 180,E1 -9985.547,E2 -9985.547} C_VEL
LIN {X 0,Y 527.923,Z 1048.869,A -85,B 0,C 180,E1 -9987.938,E2 -9987.938} C_VEL
LIN {X 0,Y 527.908,Z 1049.322,A -85,B 0,C 180,E1 -9990.543,E2 -9990.543} C_VEL
LIN {X 0,Y 527.919,Z 1048.456,A -85,B 0,C 180,E1 -9992.823,E2 -9992.823} C_VEL
LIN {X 0,Y 527.952,Z 1046.347,A -85,B 0,C 180,E1 -9995.216,E2 -9995.216} C_VEL
LIN {X 0,Y 528.045,Z 1042.438,A -85,B 0,C 180,E1 -9997.836,E2 -9997.836} C_VEL
LIN {X 0,Y 528.27,Z 1037.705,A -85,B 0,C 180,E1 -10000.139,E2 -10000.139} C_VEL
LIN {X 0,Y 528.753,Z 1030.752,A -85,B 0,C 180,E1 -10002.783,E2 -10002.783} C_VEL
LIN {X 0,Y 529.464,Z 1022.682,A -85,B 0,C 180,E1 -10005.219,E2 -10005.219} C_VEL
LIN {X 0,Y 530.591,Z 1012.631,A -85,B 0,C 180,E1 -10007.775,E2 -10007.775} C_VEL
LIN {X 0,Y 532.013,Z 1001.574,A -85,B 0,C 180,E1 -10010.117,E2 -10010.117} C_VEL
LIN {X 0,Y 533.898,Z 988.875,A -85,B 0,C 180,E1 -10012.461,E2 -10012.461} C_VEL
LIN {X 0,Y 536.192,Z 974.311,A -85,B 0,C 180,E1 -10014.748,E2 -10014.748} C_VEL
LIN {X 0,Y 538.727,Z 959.351,A -85,B 0,C 180,E1 -10016.809,E2 -10016.809} C_VEL
LIN {X 0,Y 541.681,Z 942.053,A -85,B 0,C 180,E1 -10018.862,E2 -10018.862} C_VEL
LIN {X 0,Y 544.633,Z 925.089,A -85,B 0,C 180,E1 -10020.628,E2 -10020.628} C_VEL
LIN {X 0,Y 547.95,Z 905.547,A -85,B 0,C 180,E1 -10022.383,E2 -10022.383} C_VEL
LIN {X 0,Y 550.816,Z 888.013,A -85,B 0,C 180,E1 -10023.756,E2 -10023.756} C_VEL
LIN {X 0,Y 554.233,Z 865.725,A -85,B 0,C 180,E1 -10025.262,E2 -10025.262} C_VEL
LIN {X 0,Y 556.972,Z 846.003,A -85,B 0,C 180,E1 -10026.393,E2 -10026.393} C_VEL
LIN {X 0,Y 559.952,Z 822.895,A -85,B 0,C 180,E1 -10027.511,E2 -10027.511} C_VEL
LIN {X 0,Y 562.3,Z 800.964,A -85,B 0,C 180,E1 -10028.378,E2 -10028.378} C_VEL
LIN {X 0,Y 564.529,Z 777.203,A -85,B 0,C 180,E1 -10029.136,E2 -10029.136} C_VEL
LIN {X 0,Y 566.118,Z 754.181,A -85,B 0,C 180,E1 -10029.683,E2 -10029.683} C_VEL
LIN {X 0,Y 567.209,Z 731.621,A -85,B 0,C 180,E1 -10030.081,E2 -10030.081} C_VEL
LIN {X 0,Y 574.555,Z 478.016,A -85,B 0,C 180,E1 -10033.632,E2 -10033.632} C_VEL
LIN {X 0,Y 576.001,Z 424.116,A -85,B 0,C 180,E1 -10034.411,E2 -10034.411} C_VEL
LIN {X 0,Y 564.851,Z 405.746,A -85,B 0,C 180,E1 -10035.865,E2 -10035.865} C_VEL
LIN {X 0,Y 552.746,Z 387.209,A -85,B 0,C 180,E1 -10037.531,E2 -10037.531} C_VEL
LIN {X 0,Y 540.962,Z 371.346,A -85,B 0,C 180,E1 -10039.237,E2 -10039.237} C_VEL
LIN {X 0,Y 537.745,Z 366.793,A -85,B 0,C 180,E1 -10039.731,E2 -10039.731} C_VEL
LIN {X 0,Y 534.506,Z 362.903,A -85,B 0,C 180,E1 -10040.225,E2 -10040.225} C_VEL
LIN {X 0,Y 533.406,Z 361.074,A -85,B 0,C 180,E1 -10040.406,E2 -10040.406} C_VEL
LIN {X 0,Y 530.802,Z 358.532,A -85,B 0,C 180,E1 -10040.802,E2 -10040.802} C_VEL
LIN {X 0,Y 529.655,Z 355.405,A -85,B 0,C 180,E1 -10041.022,E2 -10041.022} C_VEL
LIN {X 0,Y 529.632,Z 355.258,A -85,B 0,C 180,E1 -10044.457,E2 -10044.457} C_VEL
LIN {X 0,Y 529.686,Z 355.246,A -85,B 0,C 180,E1 -10047.837,E2 -10047.837} C_VEL
LIN {X 0,Y 529.632,Z 355.258,A -85,B 0,C 180,E1 -10051.099,E2 -10051.099} C_VEL
LIN {X 0,Y 529.632,Z 355.256,A -85,B 0,C 180,E1 -10054.624,E2 -10054.624} C_VEL
LIN {X 0,Y 529.696,Z 355.25,A -85,B 0,C 180,E1 -10057.948,E2 -10057.948} C_VEL
LIN {X 0,Y 529.631,Z 355.244,A -85,B 0,C 180,E1 -10061.28,E2 -10061.28} C_VEL
LIN {X 0,Y 529.63,Z 355.234,A -85,B 0,C 180,E1 -10064.786,E2 -10064.786} C_VEL
LIN {X 0,Y 529.678,Z 355.237,A -85,B 0,C 180,E1 -10068.015,E2 -10068.015} C_VEL
LIN {X 0,Y 529.626,Z 355.257,A -85,B 0,C 180,E1 -10071.313,E2 -10071.313} C_VEL
LIN {X 0,Y 529.646,Z 355.242,A -85,B 0,C 180,E1 -10074.692,E2 -10074.692} C_VEL
LIN {X 0,Y 529.656,Z 355.234,A -85,B 0,C 180,E1 -10077.944,E2 -10077.944} C_VEL
LIN {X 0,Y 529.627,Z 355.256,A -85,B 0,C 180,E1 -10081.19,E2 -10081.19} C_VEL
LIN {X 0,Y 529.675,Z 355.244,A -85,B 0,C 180,E1 -10084.548,E2 -10084.548} C_VEL
LIN {X 0,Y 529.631,Z 355.235,A -85,B 0,C 180,E1 -10087.812,E2 -10087.812} C_VEL
LIN {X 0,Y 529.63,Z 355.248,A -85,B 0,C 180,E1 -10091.213,E2 -10091.213} C_VEL
LIN {X 0,Y 529.695,Z 355.25,A -85,B 0,C 180,E1 -10094.54,E2 -10094.54} C_VEL
LIN {X 0,Y 529.629,Z 355.248,A -85,B 0,C 180,E1 -10097.923,E2 -10097.923} C_VEL
LIN {X 0,Y 529.627,Z 355.243,A -85,B 0,C 180,E1 -10101.449,E2 -10101.449} C_VEL
LIN {X 0,Y 529.681,Z 355.233,A -85,B 0,C 180,E1 -10104.657,E2 -10104.657} C_VEL
LIN {X 0,Y 529.623,Z 355.242,A -85,B 0,C 180,E1 -10107.926,E2 -10107.926} C_VEL
LIN {X 0,Y 529.648,Z 355.241,A -85,B 0,C 180,E1 -10111.276,E2 -10111.276} C_VEL
LIN {X 0,Y 529.652,Z 355.242,A -85,B 0,C 180,E1 -10114.496,E2 -10114.496} C_VEL
LIN {X 0,Y 529.691,Z 355.315,A -85,B 0,C 180,E1 -10116.988,E2 -10116.988} C_VEL
LIN {X 0,Y 530.949,Z 358.745,A -85,B 0,C 180,E1 -10117.601,E2 -10117.601} C_VEL
LIN {X 0,Y 535.206,Z 367.868,A -85,B 0,C 180,E1 -10119.297,E2 -10119.297} C_VEL
LIN {X 0,Y 537.106,Z 371.863,A -85,B 0,C 180,E1 -10119.961,E2 -10119.961} C_VEL
LIN {X 0,Y 550.257,Z 391.364,A -85,B 0,C 180,E1 -10121.932,E2 -10121.932} C_VEL
LIN {X 0,Y 561.965,Z 409.737,A -85,B 0,C 180,E1 -10123.571,E2 -10123.571} C_VEL
LIN {X 0,Y 574.559,Z 431.177,A -85,B 0,C 180,E1 -10125.238,E2 -10125.238} C_VEL
LIN {X 0,Y 576.111,Z 434.32,A -85,B 0,C 180,E1 -10125.444,E2 -10125.444} C_VEL
LIN {X 0,Y 568.645,Z 691.038,A -85,B 0,C 180,E1 -10129.043,E2 -10129.043} C_VEL
LIN {X 0,Y 566.414,Z 765.515,A -85,B 0,C 180,E1 -10130.103,E2 -10130.103} C_VEL
LIN {X 0,Y 564.717,Z 791.046,A -85,B 0,C 180,E1 -10130.626,E2 -10130.626} C_VEL
LIN {X 0,Y 562.818,Z 813.017,A -85,B 0,C 180,E1 -10131.233,E2 -10131.233} C_VEL
LIN {X 0,Y 560.214,Z 837.956,A -85,B 0,C 180,E1 -10132.122,E2 -10132.122} C_VEL
LIN {X 0,Y 557.737,Z 858.523,A -85,B 0,C 180,E1 -10133.025,E2 -10133.025} C_VEL
LIN {X 0,Y 554.565,Z 881.979,A -85,B 0,C 180,E1 -10134.255,E2 -10134.255} C_VEL
LIN {X 0,Y 551.741,Z 901.075,A -85,B 0,C 180,E1 -10135.442,E2 -10135.442} C_VEL
LIN {X 0,Y 548.547,Z 921.621,A -85,B 0,C 180,E1 -10136.908,E2 -10136.908} C_VEL
LIN {X 0,Y 545.28,Z 941.25,A -85,B 0,C 180,E1 -10138.554,E2 -10138.554} C_VEL
LIN {X 0,Y 542.252,Z 959.699,A -85,B 0,C 180,E1 -10140.317,E2 -10140.317} C_VEL
LIN {X 0,Y 539.291,Z 977.274,A -85,B 0,C 180,E1 -10142.265,E2 -10142.265} C_VEL
LIN {X 0,Y 536.852,Z 992.371,A -85,B 0,C 180,E1 -10144.162,E2 -10144.162} C_VEL
LIN {X 0,Y 534.341,Z 1008.597,A -85,B 0,C 180,E1 -10146.511,E2 -10146.511} C_VEL
LIN {X 0,Y 532.601,Z 1020.742,A -85,B 0,C 180,E1 -10148.525,E2 -10148.525} C_VEL
LIN {X 0,Y 530.883,Z 1034.174,A -85,B 0,C 180,E1 -10151.098,E2 -10151.098} C_VEL
LIN {X 0,Y 529.799,Z 1044.107,A -85,B 0,C 180,E1 -10153.329,E2 -10153.329} C_VEL
LIN {X 0,Y 528.929,Z 1053.828,A -85,B 0,C 180,E1 -10155.885,E2 -10155.885} C_VEL
LIN {X 0,Y 528.402,Z 1061.331,A -85,B 0,C 180,E1 -10158.318,E2 -10158.318} C_VEL
LIN {X 0,Y 528.113,Z 1067.17,A -85,B 0,C 180,E1 -10160.629,E2 -10160.629} C_VEL
LIN {X 0,Y 527.952,Z 1072.339,A -85,B 0,C 180,E1 -10163.366,E2 -10163.366} C_VEL
LIN {X 0,Y 527.922,Z 1075.177,A -85,B 0,C 180,E1 -10165.546,E2 -10165.546} C_VEL
LIN {X 0,Y 527.916,Z 1077.059,A -85,B 0,C 180,E1 -10167.938,E2 -10167.938} C_VEL
LIN {X 0,Y 527.908,Z 1077.491,A -85,B 0,C 180,E1 -10170.543,E2 -10170.543} C_VEL
LIN {X 0,Y 527.918,Z 1076.575,A -85,B 0,C 180,E1 -10172.823,E2 -10172.823} C_VEL
LIN {X 0,Y 527.935,Z 1074.249,A -85,B 0,C 180,E1 -10175.325,E2 -10175.325} C_VEL
LIN {X 0,Y 527.999,Z 1070.278,A -85,B 0,C 180,E1 -10177.837,E2 -10177.837} C_VEL
LIN {X 0,Y 528.179,Z 1065.36,A -85,B 0,C 180,E1 -10180.14,E2 -10180.14} C_VEL
LIN {X 0,Y 528.6,Z 1058.132,A -85,B 0,C 180,E1 -10182.786,E2 -10182.786} C_VEL
LIN {X 0,Y 529.214,Z 1050.2,A -85,B 0,C 180,E1 -10185.114,E2 -10185.114} C_VEL
LIN {X 0,Y 530.189,Z 1040.387,A -85,B 0,C 180,E1 -10187.562,E2 -10187.562} C_VEL
LIN {X 0,Y 531.568,Z 1028.594,A -85,B 0,C 180,E1 -10190.02,E2 -10190.02} C_VEL
LIN {X 0,Y 533.245,Z 1016.243,A -85,B 0,C 180,E1 -10192.257,E2 -10192.257} C_VEL
LIN {X 0,Y 535.463,Z 1001.15,A -85,B 0,C 180,E1 -10194.608,E2 -10194.608} C_VEL
LIN {X 0,Y 537.751,Z 986.746,A -85,B 0,C 180,E1 -10196.572,E2 -10196.572} C_VEL
LIN {X 0,Y 540.734,Z 968.504,A -85,B 0,C 180,E1 -10198.736,E2 -10198.736} C_VEL
LIN {X 0,Y 543.417,Z 952.458,A -85,B 0,C 180,E1 -10200.398,E2 -10200.398} C_VEL
LIN {X 0,Y 546.871,Z 931.728,A -85,B 0,C 180,E1 -10202.268,E2 -10202.268} C_VEL
LIN {X 0,Y 549.788,Z 913.497,A -85,B 0,C 180,E1 -10203.69,E2 -10203.69} C_VEL
LIN {X 0,Y 552.993,Z 892.795,A -85,B 0,C 180,E1 -10205.099,E2 -10205.099} C_VEL
LIN {X 0,Y 555.973,Z 871.488,A -85,B 0,C 180,E1 -10206.321,E2 -10206.321} C_VEL
LIN {X 0,Y 558.955,Z 849.03,A -85,B 0,C 180,E1 -10207.415,E2 -10207.415} C_VEL
LIN {X 0,Y 561.435,Z 826.733,A -85,B 0,C 180,E1 -10208.299,E2 -10208.299} C_VEL
LIN {X 0,Y 563.456,Z 806.196,A -85,B 0,C 180,E1 -10208.966,E2 -10208.966} C_VEL
LIN {X 0,Y 565.483,Z 780.831,A -85,B 0,C 180,E1 -10209.601,E2 -10209.601} C_VEL
LIN {X 0,Y 566.67,Z 758.726,A -85,B 0,C 180,E1 -10210.001,E2 -10210.001} C_VEL
LIN {X 0,Y 573.551,Z 518.118,A -85,B 0,C 180,E1 -10213.373,E2 -10213.373} C_VEL
LIN {X 0,Y 575.969,Z 433.715,A -85,B 0,C 180,E1 -10214.573,E2 -10214.573} C_VEL
LIN {X 0,Y 563.204,Z 411.774,A -85,B 0,C 180,E1 -10216.251,E2 -10216.251} C_VEL
LIN {X 0,Y 551.379,Z 393.108,A -85,B 0,C 180,E1 -10217.893,E2 -10217.893} C_VEL
LIN {X 0,Y 539.883,Z 375.97,A -85,B 0,C 180,E1 -10219.592,E2 -10219.592} C_VEL
LIN {X 0,Y 536.572,Z 371.047,A -85,B 0,C 180,E1 -10220.131,E2 -10220.131} C_VEL
LIN {X 0,Y 532.87,Z 362.869,A -85,B 0,C 180,E1 -10221.604,E2 -10221.604} C_VEL
LIN {X 0,Y 530.906,Z 358.662,A -85,B 0,C 180,E1 -10222.395,E2 -10222.395} C_VEL
LIN {X 0,Y 529.678,Z 355.196,A -85,B 0,C 180,E1 -10223.058,E2 -10223.058} C_VEL
LIN {X 0,Y 529.629,Z 355.228,A -85,B 0,C 180,E1 -10226.416,E2 -10226.416} C_VEL
LIN {X 0,Y 529.634,Z 355.245,A -85,B 0,C 180,E1 -10229.856,E2 -10229.856} C_VEL
LIN {X 0,Y 529.675,Z 355.236,A -85,B 0,C 180,E1 -10233.06,E2 -10233.06} C_VEL
LIN {X 0,Y 529.626,Z 355.241,A -85,B 0,C 180,E1 -10236.407,E2 -10236.407} C_VEL
LIN {X 0,Y 529.651,Z 355.236,A -85,B 0,C 180,E1 -10239.789,E2 -10239.789} C_VEL
LIN {X 0,Y 529.653,Z 355.244,A -85,B 0,C 180,E1 -10242.985,E2 -10242.985} C_VEL
LIN {X 0,Y 529.628,Z 355.256,A -85,B 0,C 180,E1 -10246.35,E2 -10246.35} C_VEL
LIN {X 0,Y 529.678,Z 355.243,A -85,B 0,C 180,E1 -10249.669,E2 -10249.669} C_VEL
LIN {X 0,Y 529.629,Z 355.231,A -85,B 0,C 180,E1 -10252.842,E2 -10252.842} C_VEL
LIN {X 0,Y 529.635,Z 355.244,A -85,B 0,C 180,E1 -10256.32,E2 -10256.32} C_VEL
LIN {X 0,Y 529.694,Z 355.25,A -85,B 0,C 180,E1 -10259.676,E2 -10259.676} C_VEL
LIN {X 0,Y 529.633,Z 355.243,A -85,B 0,C 180,E1 -10263.03,E2 -10263.03} C_VEL
LIN {X 0,Y 529.633,Z 355.233,A -85,B 0,C 180,E1 -10266.504,E2 -10266.504} C_VEL
LIN {X 0,Y 529.685,Z 355.247,A -85,B 0,C 180,E1 -10269.809,E2 -10269.809} C_VEL
LIN {X 0,Y 529.636,Z 355.254,A -85,B 0,C 180,E1 -10273.205,E2 -10273.205} C_VEL
LIN {X 0,Y 529.639,Z 355.242,A -85,B 0,C 180,E1 -10276.676,E2 -10276.676} C_VEL
LIN {X 0,Y 529.685,Z 355.232,A -85,B 0,C 180,E1 -10279.979,E2 -10279.979} C_VEL
LIN {X 0,Y 529.632,Z 355.247,A -85,B 0,C 180,E1 -10283.239,E2 -10283.239} C_VEL
LIN {X 0,Y 529.648,Z 355.249,A -85,B 0,C 180,E1 -10286.699,E2 -10286.699} C_VEL
LIN {X 0,Y 529.677,Z 355.253,A -85,B 0,C 180,E1 -10289.949,E2 -10289.949} C_VEL
LIN {X 0,Y 529.633,Z 355.256,A -85,B 0,C 180,E1 -10293.325,E2 -10293.325} C_VEL
LIN {X 0,Y 529.659,Z 355.245,A -85,B 0,C 180,E1 -10296.758,E2 -10296.758} C_VEL
LIN {X 0,Y 529.663,Z 355.433,A -85,B 0,C 180,E1 -10299.089,E2 -10299.089} C_VEL
LIN {X 0,Y 530.854,Z 358.613,A -85,B 0,C 180,E1 -10299.315,E2 -10299.315} C_VEL
LIN {X 0,Y 533.542,Z 361.167,A -85,B 0,C 180,E1 -10299.722,E2 -10299.722} C_VEL
LIN {X 0,Y 536.483,Z 365.582,A -85,B 0,C 180,E1 -10300.191,E2 -10300.191} C_VEL
LIN {X 0,Y 538.147,Z 367.586,A -85,B 0,C 180,E1 -10300.443,E2 -10300.443} C_VEL
LIN {X 0,Y 541.553,Z 371.972,A -85,B 0,C 180,E1 -10300.954,E2 -10300.954} C_VEL
LIN {X 0,Y 555.289,Z 391.02,A -85,B 0,C 180,E1 -10302.93,E2 -10302.93} C_VEL
LIN {X 0,Y 569.321,Z 412.876,A -85,B 0,C 180,E1 -10304.824,E2 -10304.824} C_VEL
LIN {X 0,Y 576.117,Z 424.672,A -85,B 0,C 180,E1 -10305.708,E2 -10305.708} C_VEL
LIN {X 0,Y 568.857,Z 672.631,A -85,B 0,C 180,E1 -10309.187,E2 -10309.187} C_VEL
LIN {X 0,Y 566.73,Z 742.589,A -85,B 0,C 180,E1 -10310.185,E2 -10310.185} C_VEL
LIN {X 0,Y 565.196,Z 767.446,A -85,B 0,C 180,E1 -10310.707,E2 -10310.707} C_VEL
LIN {X 0,Y 563.455,Z 788.732,A -85,B 0,C 180,E1 -10311.303,E2 -10311.303} C_VEL
LIN {X 0,Y 563.443,Z 788.88,A -85,B 0,C 180,E1 -10311.308,E2 -10311.308} C_VEL
LIN {X 0,Y 562,Z 796.37,A -85,B 0,C 180,E1 -10311.487,E2 -10311.487} C_VEL
LIN {X 0,Y 555.275,Z 815.1,A -85,B 0,C 180,E1 -10311.803,E2 -10311.803} C_VEL
LIN {X 0,Y 553.652,Z 822.232,A -85,B 0,C 180,E1 -10312.037,E2 -10312.037} C_VEL
LIN {X 0,Y 550.523,Z 845.759,A -85,B 0,C 180,E1 -10313.176,E2 -10313.176} C_VEL
LIN {X 0,Y 547.656,Z 865.607,A -85,B 0,C 180,E1 -10314.321,E2 -10314.321} C_VEL
LIN {X 0,Y 544.079,Z 888.017,A -85,B 0,C 180,E1 -10315.845,E2 -10315.845} C_VEL
LIN {X 0,Y 541.11,Z 905.458,A -85,B 0,C 180,E1 -10317.222,E2 -10317.222} C_VEL
LIN {X 0,Y 537.654,Z 925.027,A -85,B 0,C 180,E1 -10318.993,E2 -10318.993} C_VEL
LIN {X 0,Y 534.539,Z 942.014,A -85,B 0,C 180,E1 -10320.777,E2 -10320.777} C_VEL
LIN {X 0,Y 531.526,Z 958.931,A -85,B 0,C 180,E1 -10322.798,E2 -10322.798} C_VEL
LIN {X 0,Y 528.765,Z 974.313,A -85,B 0,C 180,E1 -10324.939,E2 -10324.939} C_VEL
LIN {X 0,Y 526.397,Z 988.598,A -85,B 0,C 180,E1 -10327.201,E2 -10327.201} C_VEL
LIN {X 0,Y 524.365,Z 1001.355,A -85,B 0,C 180,E1 -10329.577,E2 -10329.577} C_VEL
LIN {X 0,Y 522.842,Z 1012.454,A -85,B 0,C 180,E1 -10331.952,E2 -10331.952} C_VEL
LIN {X 0,Y 521.626,Z 1022.582,A -85,B 0,C 180,E1 -10334.547,E2 -10334.547} C_VEL
LIN {X 0,Y 520.874,Z 1030.34,A -85,B 0,C 180,E1 -10336.908,E2 -10336.908} C_VEL
LIN {X 0,Y 520.313,Z 1037.733,A -85,B 0,C 180,E1 -10339.711,E2 -10339.711} C_VEL
LIN {X 0,Y 520.074,Z 1042.487,A -85,B 0,C 180,E1 -10342.043,E2 -10342.043} C_VEL
LIN {X 0,Y 519.96,Z 1046.469,A -85,B 0,C 180,E1 -10344.704,E2 -10344.704} C_VEL
LIN {X 0,Y 519.922,Z 1048.615,A -85,B 0,C 180,E1 -10347.134,E2 -10347.134} C_VEL
LIN {X 0,Y 519.912,Z 1049.494,A -85,B 0,C 180,E1 -10349.339,E2 -10349.339} C_VEL
LIN {X 0,Y 519.926,Z 1049.205,A -85,B 0,C 180,E1 -10351.984,E2 -10351.984} C_VEL
LIN {X 0,Y 519.949,Z 1047.34,A -85,B 0,C 180,E1 -10354.522,E2 -10354.522} C_VEL
LIN {X 0,Y 520.01,Z 1044.465,A -85,B 0,C 180,E1 -10356.847,E2 -10356.847} C_VEL
LIN {X 0,Y 520.238,Z 1039.419,A -85,B 0,C 180,E1 -10359.626,E2 -10359.626} C_VEL
LIN {X 0,Y 520.595,Z 1033.744,A -85,B 0,C 180,E1 -10361.972,E2 -10361.972} C_VEL
LIN {X 0,Y 521.277,Z 1026.088,A -85,B 0,C 180,E1 -10364.553,E2 -10364.553} C_VEL
LIN {X 0,Y 522.266,Z 1016.952,A -85,B 0,C 180,E1 -10367.033,E2 -10367.033} C_VEL
LIN {X 0,Y 523.602,Z 1006.756,A -85,B 0,C 180,E1 -10369.407,E2 -10369.407} C_VEL
LIN {X 0,Y 525.474,Z 994.107,A -85,B 0,C 180,E1 -10371.898,E2 -10371.898} C_VEL
LIN {X 0,Y 527.471,Z 981.95,A -85,B 0,C 180,E1 -10373.978,E2 -10373.978} C_VEL
LIN {X 0,Y 530.189,Z 966.258,A -85,B 0,C 180,E1 -10376.308,E2 -10376.308} C_VEL
LIN {X 0,Y 532.851,Z 951.417,A -85,B 0,C 180,E1 -10378.221,E2 -10378.221} C_VEL
LIN {X 0,Y 536.246,Z 932.841,A -85,B 0,C 180,E1 -10380.309,E2 -10380.309} C_VEL
LIN {X 0,Y 539.252,Z 915.997,A -85,B 0,C 180,E1 -10381.948,E2 -10381.948} C_VEL
LIN {X 0,Y 542.696,Z 896.456,A -85,B 0,C 180,E1 -10383.613,E2 -10383.613} C_VEL
LIN {X 0,Y 545.928,Z 876.752,A -85,B 0,C 180,E1 -10385.045,E2 -10385.045} C_VEL
LIN {X 0,Y 549.136,Z 856.086,A -85,B 0,C 180,E1 -10386.348,E2 -10386.348} C_VEL
LIN {X 0,Y 552.102,Z 834.586,A -85,B 0,C 180,E1 -10387.482,E2 -10387.482} C_VEL
LIN {X 0,Y 554.624,Z 814.146,A -85,B 0,C 180,E1 -10388.395,E2 -10388.395} C_VEL
LIN {X 0,Y 557.213,Z 789.283,A -85,B 0,C 180,E1 -10389.296,E2 -10389.296} C_VEL
LIN {X 0,Y 559.037,Z 767.809,A -85,B 0,C 180,E1 -10389.903,E2 -10389.903} C_VEL
LIN {X 0,Y 560.626,Z 743.016,A -85,B 0,C 180,E1 -10390.429,E2 -10390.429} C_VEL
LIN {X 0,Y 562.769,Z 675.99,A -85,B 0,C 180,E1 -10391.395,E2 -10391.395} C_VEL
LIN {X 0,Y 570.308,Z 429.687,A -85,B 0,C 180,E1 -10394.88,E2 -10394.88} C_VEL
LIN {X 0,Y 570.208,Z 427.548,A -85,B 0,C 180,E1 -10394.928,E2 -10394.928} C_VEL
LIN {X 0,Y 560.004,Z 410.695,A -85,B 0,C 180,E1 -10396.291,E2 -10396.291} C_VEL
LIN {X 0,Y 548.527,Z 393.049,A -85,B 0,C 180,E1 -10397.905,E2 -10397.905} C_VEL
LIN {X 0,Y 537.145,Z 377.608,A -85,B 0,C 180,E1 -10399.587,E2 -10399.587} C_VEL
LIN {X 0,Y 532.565,Z 371.653,A -85,B 0,C 180,E1 -10400.296,E2 -10400.296} C_VEL
LIN {X 0,Y 529.479,Z 367.472,A -85,B 0,C 180,E1 -10400.79,E2 -10400.79} C_VEL
LIN {X 0,Y 526.535,Z 363.84,A -85,B 0,C 180,E1 -10401.265,E2 -10401.265} C_VEL
LIN {X 0,Y 525.554,Z 362.113,A -85,B 0,C 180,E1 -10401.436,E2 -10401.436} C_VEL
LIN {X 0,Y 522.857,Z 359.43,A -85,B 0,C 180,E1 -10401.869,E2 -10401.869} C_VEL
LIN {X 0,Y 521.722,Z 356.292,A -85,B 0,C 180,E1 -10402.098,E2 -10402.098} C_VEL
LIN {X 0,Y 521.723,Z 356.228,A -85,B 0,C 180,E1 -10405.438,E2 -10405.438} C_VEL
LIN {X 0,Y 521.685,Z 356.231,A -85,B 0,C 180,E1 -10408.741,E2 -10408.741} C_VEL
LIN {X 0,Y 521.734,Z 356.223,A -85,B 0,C 180,E1 -10412.067,E2 -10412.067} C_VEL
LIN {X 0,Y 521.708,Z 356.232,A -85,B 0,C 180,E1 -10415.424,E2 -10415.424} C_VEL
LIN {X 0,Y 521.691,Z 356.245,A -85,B 0,C 180,E1 -10418.762,E2 -10418.762} C_VEL
LIN {X 0,Y 521.742,Z 356.242,A -85,B 0,C 180,E1 -10422.144,E2 -10422.144} C_VEL
LIN {X 0,Y 521.694,Z 356.228,A -85,B 0,C 180,E1 -10425.459,E2 -10425.459} C_VEL
LIN {X 0,Y 521.687,Z 356.221,A -85,B 0,C 180,E1 -10428.95,E2 -10428.95} C_VEL
LIN {X 0,Y 521.749,Z 356.231,A -85,B 0,C 180,E1 -10432.291,E2 -10432.291} C_VEL
LIN {X 0,Y 521.696,Z 356.242,A -85,B 0,C 180,E1 -10435.603,E2 -10435.603} C_VEL
LIN {X 0,Y 521.687,Z 356.227,A -85,B 0,C 180,E1 -10439.121,E2 -10439.121} C_VEL
LIN {X 0,Y 521.739,Z 356.218,A -85,B 0,C 180,E1 -10442.416,E2 -10442.416} C_VEL
LIN {X 0,Y 521.699,Z 356.248,A -85,B 0,C 180,E1 -10445.83,E2 -10445.83} C_VEL
LIN {X 0,Y 521.689,Z 356.243,A -85,B 0,C 180,E1 -10449.265,E2 -10449.265} C_VEL
LIN {X 0,Y 521.741,Z 356.219,A -85,B 0,C 180,E1 -10452.62,E2 -10452.62} C_VEL
LIN {X 0,Y 521.689,Z 356.231,A -85,B 0,C 180,E1 -10455.814,E2 -10455.814} C_VEL
LIN {X 0,Y 521.691,Z 356.24,A -85,B 0,C 180,E1 -10459.365,E2 -10459.365} C_VEL
LIN {X 0,Y 521.758,Z 356.239,A -85,B 0,C 180,E1 -10462.656,E2 -10462.656} C_VEL
LIN {X 0,Y 521.693,Z 356.244,A -85,B 0,C 180,E1 -10466.034,E2 -10466.034} C_VEL
LIN {X 0,Y 521.695,Z 356.248,A -85,B 0,C 180,E1 -10469.524,E2 -10469.524} C_VEL
LIN {X 0,Y 521.746,Z 356.244,A -85,B 0,C 180,E1 -10472.844,E2 -10472.844} C_VEL
LIN {X 0,Y 521.705,Z 356.392,A -85,B 0,C 180,E1 -10475.999,E2 -10475.999} C_VEL
LIN {X 0,Y 522.988,Z 359.66,A -85,B 0,C 180,E1 -10476.62,E2 -10476.62} C_VEL
LIN {X 0,Y 523.854,Z 361.305,A -85,B 0,C 180,E1 -10476.959,E2 -10476.959} C_VEL
LIN {X 0,Y 528.334,Z 371.205,A -85,B 0,C 180,E1 -10478.805,E2 -10478.805} C_VEL
LIN {X 0,Y 537.971,Z 385.05,A -85,B 0,C 180,E1 -10480.336,E2 -10480.336} C_VEL
LIN {X 0,Y 549.89,Z 402.941,A -85,B 0,C 180,E1 -10482.111,E2 -10482.111} C_VEL
LIN {X 0,Y 563.303,Z 424.978,A -85,B 0,C 180,E1 -10483.987,E2 -10483.987} C_VEL
LIN {X 0,Y 570.304,Z 437.414,A -85,B 0,C 180,E1 -10484.924,E2 -10484.924} C_VEL
LIN {X 0,Y 562.538,Z 693.139,A -85,B 0,C 180,E1 -10488.539,E2 -10488.539} C_VEL
LIN {X 0,Y 560.272,Z 765.425,A -85,B 0,C 180,E1 -10489.578,E2 -10489.578} C_VEL
LIN {X 0,Y 558.521,Z 790.842,A -85,B 0,C 180,E1 -10490.103,E2 -10490.103} C_VEL
LIN {X 0,Y 556.545,Z 812.846,A -85,B 0,C 180,E1 -10490.714,E2 -10490.714} C_VEL
LIN {X 0,Y 553.834,Z 837.746,A -85,B 0,C 180,E1 -10491.607,E2 -10491.607} C_VEL
LIN {X 0,Y 551.257,Z 858.312,A -85,B 0,C 180,E1 -10492.516,E2 -10492.516} C_VEL
LIN {X 0,Y 547.931,Z 881.901,A -85,B 0,C 180,E1 -10493.764,E2 -10493.764} C_VEL
LIN {X 0,Y 545.01,Z 900.86,A -85,B 0,C 180,E1 -10494.954,E2 -10494.954} C_VEL
LIN {X 0,Y 541.67,Z 921.448,A -85,B 0,C 180,E1 -10496.437,E2 -10496.437} C_VEL
LIN {X 0,Y 538.246,Z 941.074,A -85,B 0,C 180,E1 -10498.099,E2 -10498.099} C_VEL
LIN {X 0,Y 535.006,Z 959.891,A -85,B 0,C 180,E1 -10499.919,E2 -10499.919} C_VEL
LIN {X 0,Y 531.97,Z 977.055,A -85,B 0,C 180,E1 -10501.85,E2 -10501.85} C_VEL
LIN {X 0,Y 529.365,Z 992.324,A -85,B 0,C 180,E1 -10503.793,E2 -10503.793} C_VEL
LIN {X 0,Y 526.748,Z 1008.378,A -85,B 0,C 180,E1 -10506.151,E2 -10506.151} C_VEL
LIN {X 0,Y 524.899,Z 1020.522,A -85,B 0,C 180,E1 -10508.194,E2 -10508.194} C_VEL
LIN {X 0,Y 523.079,Z 1033.954,A -85,B 0,C 180,E1 -10510.805,E2 -10510.805} C_VEL
LIN {X 0,Y 521.927,Z 1043.888,A -85,B 0,C 180,E1 -10513.07,E2 -10513.07} C_VEL
LIN {X 0,Y 520.998,Z 1053.609,A -85,B 0,C 180,E1 -10515.666,E2 -10515.666} C_VEL
LIN {X 0,Y 520.436,Z 1061.114,A -85,B 0,C 180,E1 -10518.137,E2 -10518.137} C_VEL
LIN {X 0,Y 520.118,Z 1067.212,A -85,B 0,C 180,E1 -10520.595,E2 -10520.595} C_VEL
LIN {X 0,Y 519.957,Z 1072.124,A -85,B 0,C 180,E1 -10523.263,E2 -10523.263} C_VEL
LIN {X 0,Y 519.925,Z 1074.963,A -85,B 0,C 180,E1 -10525.478,E2 -10525.478} C_VEL
LIN {X 0,Y 519.918,Z 1076.846,A -85,B 0,C 180,E1 -10527.906,E2 -10527.906} C_VEL
LIN {X 0,Y 519.911,Z 1077.278,A -85,B 0,C 180,E1 -10530.551,E2 -10530.551} C_VEL
LIN {X 0,Y 519.922,Z 1076.361,A -85,B 0,C 180,E1 -10532.866,E2 -10532.866} C_VEL
LIN {X 0,Y 519.938,Z 1074.035,A -85,B 0,C 180,E1 -10535.407,E2 -10535.407} C_VEL
LIN {X 0,Y 520.01,Z 1069.979,A -85,B 0,C 180,E1 -10538.002,E2 -10538.002} C_VEL
LIN {X 0,Y 520.199,Z 1065.144,A -85,B 0,C 180,E1 -10540.297,E2 -10540.297} C_VEL
LIN {X 0,Y 520.65,Z 1057.914,A -85,B 0,C 180,E1 -10542.985,E2 -10542.985} C_VEL
LIN {X 0,Y 521.303,Z 1049.981,A -85,B 0,C 180,E1 -10545.349,E2 -10545.349} C_VEL
LIN {X 0,Y 522.34,Z 1040.167,A -85,B 0,C 180,E1 -10547.835,E2 -10547.835} C_VEL
LIN {X 0,Y 523.8,Z 1028.372,A -85,B 0,C 180,E1 -10550.33,E2 -10550.33} C_VEL
LIN {X 0,Y 525.589,Z 1016.02,A -85,B 0,C 180,E1 -10552.599,E2 -10552.599} C_VEL
LIN {X 0,Y 527.931,Z 1000.926,A -85,B 0,C 180,E1 -10554.983,E2 -10554.983} C_VEL
LIN {X 0,Y 530.258,Z 987.015,A -85,B 0,C 180,E1 -10556.908,E2 -10556.908} C_VEL
LIN {X 0,Y 533.482,Z 968.28,A -85,B 0,C 180,E1 -10559.164,E2 -10559.164} C_VEL
LIN {X 0,Y 536.409,Z 951.675,A -85,B 0,C 180,E1 -10560.9,E2 -10560.9} C_VEL
LIN {X 0,Y 540.032,Z 930.775,A -85,B 0,C 180,E1 -10562.796,E2 -10562.796} C_VEL
LIN {X 0,Y 542.962,Z 913.273,A -85,B 0,C 180,E1 -10564.171,E2 -10564.171} C_VEL
LIN {X 0,Y 546.315,Z 892.572,A -85,B 0,C 180,E1 -10565.592,E2 -10565.592} C_VEL
LIN {X 0,Y 549.329,Z 871.963,A -85,B 0,C 180,E1 -10566.787,E2 -10566.787} C_VEL
LIN {X 0,Y 552.32,Z 850.284,A -85,B 0,C 180,E1 -10567.858,E2 -10567.858} C_VEL
LIN {X 0,Y 555.024,Z 827.305,A -85,B 0,C 180,E1 -10568.788,E2 -10568.788} C_VEL
LIN {X 0,Y 557.104,Z 807.022,A -85,B 0,C 180,E1 -10569.456,E2 -10569.456} C_VEL
LIN {X 0,Y 559.209,Z 782.248,A -85,B 0,C 180,E1 -10570.092,E2 -10570.092} C_VEL
LIN {X 0,Y 560.51,Z 759.189,A -85,B 0,C 180,E1 -10570.517,E2 -10570.517} C_VEL
LIN {X 0,Y 567.648,Z 520.633,A -85,B 0,C 180,E1 -10573.891,E2 -10573.891} C_VEL
LIN {X 0,Y 570.109,Z 436.956,A -85,B 0,C 180,E1 -10575.095,E2 -10575.095} C_VEL
LIN {X 0,Y 557.385,Z 415.087,A -85,B 0,C 180,E1 -10576.814,E2 -10576.814} C_VEL
LIN {X 0,Y 544.543,Z 394.786,A -85,B 0,C 180,E1 -10578.656,E2 -10578.656} C_VEL
LIN {X 0,Y 532.089,Z 376.608,A -85,B 0,C 180,E1 -10580.568,E2 -10580.568} C_VEL
LIN {X 0,Y 527.961,Z 370.501,A -85,B 0,C 180,E1 -10581.286,E2 -10581.286} C_VEL
LIN {X 0,Y 523.288,Z 360.019,A -85,B 0,C 180,E1 -10583.268,E2 -10583.268} C_VEL
LIN {X 0,Y 521.729,Z 356.507,A -85,B 0,C 180,E1 -10583.959,E2 -10583.959} C_VEL
LIN {X 0,Y 521.679,Z 356.173,A -85,B 0,C 180,E1 -10584.17,E2 -10584.17} C_VEL
LIN {X 0,Y 521.716,Z 356.238,A -85,B 0,C 180,E1 -10587.545,E2 -10587.545} C_VEL
LIN {X 0,Y 521.713,Z 356.241,A -85,B 0,C 180,E1 -10590.743,E2 -10590.743} C_VEL
LIN {X 0,Y 521.692,Z 356.246,A -85,B 0,C 180,E1 -10594.088,E2 -10594.088} C_VEL
LIN {X 0,Y 521.744,Z 356.237,A -85,B 0,C 180,E1 -10597.476,E2 -10597.476} C_VEL
LIN {X 0,Y 521.698,Z 356.234,A -85,B 0,C 180,E1 -10600.752,E2 -10600.752} C_VEL
LIN {X 0,Y 521.689,Z 356.226,A -85,B 0,C 180,E1 -10604.207,E2 -10604.207} C_VEL
LIN {X 0,Y 521.744,Z 356.223,A -85,B 0,C 180,E1 -10607.493,E2 -10607.493} C_VEL
LIN {X 0,Y 521.695,Z 356.245,A -85,B 0,C 180,E1 -10610.846,E2 -10610.846} C_VEL
LIN {X 0,Y 521.693,Z 356.244,A -85,B 0,C 180,E1 -10614.39,E2 -10614.39} C_VEL
LIN {X 0,Y 521.742,Z 356.217,A -85,B 0,C 180,E1 -10617.693,E2 -10617.693} C_VEL
LIN {X 0,Y 521.693,Z 356.236,A -85,B 0,C 180,E1 -10620.988,E2 -10620.988} C_VEL
LIN {X 0,Y 521.695,Z 356.246,A -85,B 0,C 180,E1 -10624.507,E2 -10624.507} C_VEL
LIN {X 0,Y 521.753,Z 356.222,A -85,B 0,C 180,E1 -10627.82,E2 -10627.82} C_VEL
LIN {X 0,Y 521.694,Z 356.222,A -85,B 0,C 180,E1 -10631.162,E2 -10631.162} C_VEL
LIN {X 0,Y 521.697,Z 356.236,A -85,B 0,C 180,E1 -10634.655,E2 -10634.655} C_VEL
LIN {X 0,Y 521.749,Z 356.241,A -85,B 0,C 180,E1 -10637.972,E2 -10637.972} C_VEL
LIN {X 0,Y 521.7,Z 356.24,A -85,B 0,C 180,E1 -10641.356,E2 -10641.356} C_VEL
LIN {X 0,Y 521.699,Z 356.231,A -85,B 0,C 180,E1 -10644.818,E2 -10644.818} C_VEL
LIN {X 0,Y 521.756,Z 356.221,A -85,B 0,C 180,E1 -10648.171,E2 -10648.171} C_VEL
LIN {X 0,Y 521.696,Z 356.226,A -85,B 0,C 180,E1 -10651.472,E2 -10651.472} C_VEL
LIN {X 0,Y 521.702,Z 356.229,A -85,B 0,C 180,E1 -10654.964,E2 -10654.964} C_VEL
LIN {X 0,Y 521.753,Z 356.422,A -85,B 0,C 180,E1 -10658.02,E2 -10658.02} C_VEL
LIN {X 0,Y 522.968,Z 359.58,A -85,B 0,C 180,E1 -10658.26,E2 -10658.26} C_VEL
LIN {X 0,Y 525.994,Z 362.749,A -85,B 0,C 180,E1 -10658.748,E2 -10658.748} C_VEL
LIN {X 0,Y 528.594,Z 366.654,A -85,B 0,C 180,E1 -10659.183,E2 -10659.183} C_VEL
LIN {X 0,Y 530.453,Z 368.663,A -85,B 0,C 180,E1 -10659.473,E2 -10659.473} C_VEL
LIN {X 0,Y 542.562,Z 384.965,A -85,B 0,C 180,E1 -10661.335,E2 -10661.335} C_VEL
LIN {X 0,Y 552.616,Z 399.077,A -85,B 0,C 180,E1 -10662.781,E2 -10662.781} C_VEL
LIN {X 0,Y 566.869,Z 421.891,A -85,B 0,C 180,E1 -10664.732,E2 -10664.732} C_VEL
LIN {X 0,Y 570.314,Z 428.167,A -85,B 0,C 180,E1 -10665.193,E2 -10665.193} C_VEL
LIN {X 0,Y 562.725,Z 676.252,A -85,B 0,C 180,E1 -10668.702,E2 -10668.702} C_VEL
LIN {X 0,Y 560.597,Z 743.042,A -85,B 0,C 180,E1 -10669.665,E2 -10669.665} C_VEL
LIN {X 0,Y 559.005,Z 767.805,A -85,B 0,C 180,E1 -10670.19,E2 -10670.19} C_VEL
LIN {X 0,Y 557.19,Z 789.175,A -85,B 0,C 180,E1 -10670.793,E2 -10670.793} C_VEL
LIN {X 0,Y 554.665,Z 813.576,A -85,B 0,C 180,E1 -10671.675,E2 -10671.675} C_VEL
LIN {X 0,Y 553.652,Z 822.232,A -85,B 0,C 180,E1 -10672.037,E2 -10672.037} C_VEL
LIN {X 0,Y 551.978,Z 829.438,A -85,B 0,C 180,E1 -10672.291,E2 -10672.291} C_VEL
LIN {X 0,Y 544.661,Z 847.494,A -85,B 0,C 180,E1 -10672.814,E2 -10672.814} C_VEL
LIN {X 0,Y 542.897,Z 854.394,A -85,B 0,C 180,E1 -10673.128,E2 -10673.128} C_VEL
LIN {X 0,Y 539.471,Z 875.807,A -85,B 0,C 180,E1 -10674.475,E2 -10674.475} C_VEL
LIN {X 0,Y 536.338,Z 894.164,A -85,B 0,C 180,E1 -10675.808,E2 -10675.808} C_VEL
LIN {X 0,Y 532.488,Z 915.26,A -85,B 0,C 180,E1 -10677.592,E2 -10677.592} C_VEL
LIN {X 0,Y 529.385,Z 931.853,A -85,B 0,C 180,E1 -10679.212,E2 -10679.212} C_VEL
LIN {X 0,Y 525.763,Z 950.946,A -85,B 0,C 180,E1 -10681.364,E2 -10681.364} C_VEL
LIN {X 0,Y 522.935,Z 965.843,A -85,B 0,C 180,E1 -10683.299,E2 -10683.299} C_VEL
LIN {X 0,Y 520.014,Z 981.904,A -85,B 0,C 180,E1 -10685.702,E2 -10685.702} C_VEL
LIN {X 0,Y 517.931,Z 993.846,A -85,B 0,C 180,E1 -10687.766,E2 -10687.766} C_VEL
LIN {X 0,Y 515.933,Z 1006.586,A -85,B 0,C 180,E1 -10690.293,E2 -10690.293} C_VEL
LIN {X 0,Y 514.494,Z 1016.819,A -85,B 0,C 180,E1 -10692.702,E2 -10692.702} C_VEL
LIN {X 0,Y 513.42,Z 1025.991,A -85,B 0,C 180,E1 -10695.219,E2 -10695.219} C_VEL
LIN {X 0,Y 512.677,Z 1033.722,A -85,B 0,C 180,E1 -10697.841,E2 -10697.841} C_VEL
LIN {X 0,Y 512.273,Z 1039.435,A -85,B 0,C 180,E1 -10700.223,E2 -10700.223} C_VEL
LIN {X 0,Y 512.037,Z 1044.553,A -85,B 0,C 180,E1 -10703.046,E2 -10703.046} C_VEL
LIN {X 0,Y 511.955,Z 1047.463,A -85,B 0,C 180,E1 -10705.407,E2 -10705.407} C_VEL
LIN {X 0,Y 511.93,Z 1049.297,A -85,B 0,C 180,E1 -10707.873,E2 -10707.873} C_VEL
LIN {X 0,Y 511.914,Z 1049.748,A -85,B 0,C 180,E1 -10710.56,E2 -10710.56} C_VEL
LIN {X 0,Y 511.927,Z 1048.883,A -85,B 0,C 180,E1 -10712.911,E2 -10712.911} C_VEL
LIN {X 0,Y 511.964,Z 1046.774,A -85,B 0,C 180,E1 -10715.379,E2 -10715.379} C_VEL
LIN {X 0,Y 512.093,Z 1042.78,A -85,B 0,C 180,E1 -10718.13,E2 -10718.13} C_VEL
LIN {X 0,Y 512.348,Z 1038.134,A -85,B 0,C 180,E1 -10720.457,E2 -10720.457} C_VEL
LIN {X 0,Y 512.909,Z 1031.183,A -85,B 0,C 180,E1 -10723.184,E2 -10723.184} C_VEL
LIN {X 0,Y 513.731,Z 1023.114,A -85,B 0,C 180,E1 -10725.696,E2 -10725.696} C_VEL
LIN {X 0,Y 515.017,Z 1013.064,A -85,B 0,C 180,E1 -10728.332,E2 -10728.332} C_VEL
LIN {X 0,Y 516.664,Z 1001.669,A -85,B 0,C 180,E1 -10730.813,E2 -10730.813} C_VEL
LIN {X 0,Y 518.854,Z 988.66,A -85,B 0,C 180,E1 -10733.27,E2 -10733.27} C_VEL
LIN {X 0,Y 521.368,Z 974.352,A -85,B 0,C 180,E1 -10735.563,E2 -10735.563} C_VEL
LIN {X 0,Y 524.339,Z 958.665,A -85,B 0,C 180,E1 -10737.769,E2 -10737.769} C_VEL
LIN {X 0,Y 527.455,Z 941.981,A -85,B 0,C 180,E1 -10739.78,E2 -10739.78} C_VEL
LIN {X 0,Y 530.84,Z 924.448,A -85,B 0,C 180,E1 -10741.637,E2 -10741.637} C_VEL
LIN {X 0,Y 534.348,Z 905.31,A -85,B 0,C 180,E1 -10743.377,E2 -10743.377} C_VEL
LIN {X 0,Y 537.58,Z 887.125,A -85,B 0,C 180,E1 -10744.821,E2 -10744.821} C_VEL
LIN {X 0,Y 541.195,Z 865.248,A -85,B 0,C 180,E1 -10746.309,E2 -10746.309} C_VEL
LIN {X 0,Y 544.031,Z 846.419,A -85,B 0,C 180,E1 -10747.404,E2 -10747.404} C_VEL
LIN {X 0,Y 547.252,Z 823.306,A -85,B 0,C 180,E1 -10748.539,E2 -10748.539} C_VEL
LIN {X 0,Y 549.596,Z 803.068,A -85,B 0,C 180,E1 -10749.357,E2 -10749.357} C_VEL
LIN {X 0,Y 551.817,Z 781.159,A -85,B 0,C 180,E1 -10750.082,E2 -10750.082} C_VEL
LIN {X 0,Y 553.768,Z 756.353,A -85,B 0,C 180,E1 -10750.705,E2 -10750.705} C_VEL
LIN {X 0,Y 554.935,Z 734.651,A -85,B 0,C 180,E1 -10751.103,E2 -10751.103} C_VEL
LIN {X 0,Y 562.838,Z 485.371,A -85,B 0,C 180,E1 -10754.657,E2 -10754.657} C_VEL
LIN {X 0,Y 564.463,Z 430.99,A -85,B 0,C 180,E1 -10755.454,E2 -10755.454} C_VEL
LIN {X 0,Y 553.558,Z 412.922,A -85,B 0,C 180,E1 -10756.956,E2 -10756.956} C_VEL
LIN {X 0,Y 543.887,Z 398.322,A -85,B 0,C 180,E1 -10758.349,E2 -10758.349} C_VEL
LIN {X 0,Y 533.334,Z 383.837,A -85,B 0,C 180,E1 -10759.945,E2 -10759.945} C_VEL
LIN {X 0,Y 525.593,Z 373.687,A -85,B 0,C 180,E1 -10761.182,E2 -10761.182} C_VEL
LIN {X 0,Y 522.372,Z 369.242,A -85,B 0,C 180,E1 -10761.723,E2 -10761.723} C_VEL
LIN {X 0,Y 518.865,Z 365.093,A -85,B 0,C 180,E1 -10762.312,E2 -10762.312} C_VEL
LIN {X 0,Y 517.686,Z 363.16,A -85,B 0,C 180,E1 -10762.525,E2 -10762.525} C_VEL
LIN {X 0,Y 514.996,Z 360.607,A -85,B 0,C 180,E1 -10762.978,E2 -10762.978} C_VEL
LIN {X 0,Y 513.817,Z 357.54,A -85,B 0,C 180,E1 -10763.224,E2 -10763.224} C_VEL
LIN {X 0,Y 513.777,Z 357.22,A -85,B 0,C 180,E1 -10763.311,E2 -10763.311} C_VEL
LIN {X 0,Y 513.748,Z 357.229,A -85,B 0,C 180,E1 -10766.712,E2 -10766.712} C_VEL
LIN {X 0,Y 513.788,Z 357.225,A -85,B 0,C 180,E1 -10770.118,E2 -10770.118} C_VEL
LIN {X 0,Y 513.76,Z 357.219,A -85,B 0,C 180,E1 -10773.293,E2 -10773.293} C_VEL
LIN {X 0,Y 513.751,Z 357.216,A -85,B 0,C 180,E1 -10776.728,E2 -10776.728} C_VEL
LIN {X 0,Y 513.806,Z 357.207,A -85,B 0,C 180,E1 -10780.042,E2 -10780.042} C_VEL
LIN {X 0,Y 513.756,Z 357.226,A -85,B 0,C 180,E1 -10783.375,E2 -10783.375} C_VEL
LIN {X 0,Y 513.754,Z 357.234,A -85,B 0,C 180,E1 -10786.838,E2 -10786.838} C_VEL
LIN {X 0,Y 513.801,Z 357.215,A -85,B 0,C 180,E1 -10790.252,E2 -10790.252} C_VEL
LIN {X 0,Y 513.751,Z 357.212,A -85,B 0,C 180,E1 -10793.518,E2 -10793.518} C_VEL
LIN {X 0,Y 513.753,Z 357.229,A -85,B 0,C 180,E1 -10796.988,E2 -10796.988} C_VEL
LIN {X 0,Y 513.817,Z 357.226,A -85,B 0,C 180,E1 -10800.334,E2 -10800.334} C_VEL
LIN {X 0,Y 513.758,Z 357.21,A -85,B 0,C 180,E1 -10803.794,E2 -10803.794} C_VEL
LIN {X 0,Y 513.746,Z 357.214,A -85,B 0,C 180,E1 -10807.268,E2 -10807.268} C_VEL
LIN {X 0,Y 513.803,Z 357.226,A -85,B 0,C 180,E1 -10810.541,E2 -10810.541} C_VEL
LIN {X 0,Y 513.759,Z 357.23,A -85,B 0,C 180,E1 -10813.965,E2 -10813.965} C_VEL
LIN {X 0,Y 513.747,Z 357.219,A -85,B 0,C 180,E1 -10817.441,E2 -10817.441} C_VEL
LIN {X 0,Y 513.804,Z 357.206,A -85,B 0,C 180,E1 -10820.743,E2 -10820.743} C_VEL
LIN {X 0,Y 513.752,Z 357.218,A -85,B 0,C 180,E1 -10824.002,E2 -10824.002} C_VEL
LIN {X 0,Y 513.754,Z 357.221,A -85,B 0,C 180,E1 -10827.469,E2 -10827.469} C_VEL
LIN {X 0,Y 513.816,Z 357.215,A -85,B 0,C 180,E1 -10830.784,E2 -10830.784} C_VEL
LIN {X 0,Y 513.753,Z 357.222,A -85,B 0,C 180,E1 -10834.192,E2 -10834.192} C_VEL
LIN {X 0,Y 513.815,Z 357.318,A -85,B 0,C 180,E1 -10834.948,E2 -10834.948} C_VEL
LIN {X 0,Y 515.08,Z 360.751,A -85,B 0,C 180,E1 -10835.618,E2 -10835.618} C_VEL
LIN {X 0,Y 516.129,Z 363.006,A -85,B 0,C 180,E1 -10836.082,E2 -10836.082} C_VEL
LIN {X 0,Y 518.035,Z 366.966,A -85,B 0,C 180,E1 -10836.89,E2 -10836.89} C_VEL
LIN {X 0,Y 519.966,Z 371.039,A -85,B 0,C 180,E1 -10837.647,E2 -10837.647} C_VEL
LIN {X 0,Y 533.175,Z 389.678,A -85,B 0,C 180,E1 -10839.824,E2 -10839.824} C_VEL
LIN {X 0,Y 546.46,Z 410.013,A -85,B 0,C 180,E1 -10841.85,E2 -10841.85} C_VEL
LIN {X 0,Y 559.045,Z 430.902,A -85,B 0,C 180,E1 -10843.643,E2 -10843.643} C_VEL
LIN {X 0,Y 564.537,Z 440.801,A -85,B 0,C 180,E1 -10844.397,E2 -10844.397} C_VEL
LIN {X 0,Y 556.474,Z 695.241,A -85,B 0,C 180,E1 -10848.024,E2 -10848.024} C_VEL
LIN {X 0,Y 554.179,Z 765.337,A -85,B 0,C 180,E1 -10849.041,E2 -10849.041} C_VEL
LIN {X 0,Y 552.363,Z 790.769,A -85,B 0,C 180,E1 -10849.571,E2 -10849.571} C_VEL
LIN {X 0,Y 550.316,Z 812.732,A -85,B 0,C 180,E1 -10850.185,E2 -10850.185} C_VEL
LIN {X 0,Y 547.502,Z 837.537,A -85,B 0,C 180,E1 -10851.08,E2 -10851.08} C_VEL
LIN {X 0,Y 544.824,Z 858.101,A -85,B 0,C 180,E1 -10851.995,E2 -10851.995} C_VEL
LIN {X 0,Y 541.383,Z 881.552,A -85,B 0,C 180,E1 -10853.244,E2 -10853.244} C_VEL
LIN {X 0,Y 538.318,Z 900.645,A -85,B 0,C 180,E1 -10854.452,E2 -10854.452} C_VEL
LIN {X 0,Y 534.839,Z 921.231,A -85,B 0,C 180,E1 -10855.95,E2 -10855.95} C_VEL
LIN {X 0,Y 531.268,Z 940.816,A -85,B 0,C 180,E1 -10857.625,E2 -10857.625} C_VEL
LIN {X 0,Y 527.956,Z 959.073,A -85,B 0,C 180,E1 -10859.408,E2 -10859.408} C_VEL
LIN {X 0,Y 524.678,Z 976.836,A -85,B 0,C 180,E1 -10861.423,E2 -10861.423} C_VEL
LIN {X 0,Y 521.962,Z 991.932,A -85,B 0,C 180,E1 -10863.368,E2 -10863.368} C_VEL
LIN {X 0,Y 519.173,Z 1008.158,A -85,B 0,C 180,E1 -10865.781,E2 -10865.781} C_VEL
LIN {X 0,Y 517.12,Z 1020.945,A -85,B 0,C 180,E1 -10867.969,E2 -10867.969} C_VEL
LIN {X 0,Y 515.217,Z 1034.257,A -85,B 0,C 180,E1 -10870.618,E2 -10870.618} C_VEL
LIN {X 0,Y 514.009,Z 1044.135,A -85,B 0,C 180,E1 -10872.918,E2 -10872.918} C_VEL
LIN {X 0,Y 513.002,Z 1054.109,A -85,B 0,C 180,E1 -10875.668,E2 -10875.668} C_VEL
LIN {X 0,Y 512.451,Z 1061.205,A -85,B 0,C 180,E1 -10878.063,E2 -10878.063} C_VEL
LIN {X 0,Y 512.107,Z 1067.512,A -85,B 0,C 180,E1 -10880.674,E2 -10880.674} C_VEL
LIN {X 0,Y 511.957,Z 1072.072,A -85,B 0,C 180,E1 -10883.27,E2 -10883.27} C_VEL
LIN {X 0,Y 511.925,Z 1074.865,A -85,B 0,C 180,E1 -10885.519,E2 -10885.519} C_VEL
LIN {X 0,Y 511.916,Z 1076.769,A -85,B 0,C 180,E1 -10888.097,E2 -10888.097} C_VEL
LIN {X 0,Y 511.915,Z 1077.042,A -85,B 0,C 180,E1 -10890.671,E2 -10890.671} C_VEL
LIN {X 0,Y 511.925,Z 1076.147,A -85,B 0,C 180,E1 -10892.911,E2 -10892.911} C_VEL
LIN {X 0,Y 511.939,Z 1073.82,A -85,B 0,C 180,E1 -10895.492,E2 -10895.492} C_VEL
LIN {X 0,Y 512.017,Z 1069.847,A -85,B 0,C 180,E1 -10898.083,E2 -10898.083} C_VEL
LIN {X 0,Y 512.206,Z 1065.186,A -85,B 0,C 180,E1 -10900.346,E2 -10900.346} C_VEL
LIN {X 0,Y 512.648,Z 1058.412,A -85,B 0,C 180,E1 -10902.962,E2 -10902.962} C_VEL
LIN {X 0,Y 513.357,Z 1050.172,A -85,B 0,C 180,E1 -10905.476,E2 -10905.476} C_VEL
LIN {X 0,Y 514.322,Z 1041.343,A -85,B 0,C 180,E1 -10907.771,E2 -10907.771} C_VEL
LIN {X 0,Y 515.892,Z 1029.312,A -85,B 0,C 180,E1 -10910.418,E2 -10910.418} C_VEL
LIN {X 0,Y 517.627,Z 1017.727,A -85,B 0,C 180,E1 -10912.607,E2 -10912.607} C_VEL
LIN {X 0,Y 520.036,Z 1003.041,A -85,B 0,C 180,E1 -10915.024,E2 -10915.024} C_VEL
LIN {X 0,Y 522.562,Z 988.5,A -85,B 0,C 180,E1 -10917.09,E2 -10917.09} C_VEL
LIN {X 0,Y 525.583,Z 971.986,A -85,B 0,C 180,E1 -10919.164,E2 -10919.164} C_VEL
LIN {X 0,Y 528.911,Z 953.691,A -85,B 0,C 180,E1 -10921.134,E2 -10921.134} C_VEL
LIN {X 0,Y 532.388,Z 934.901,A -85,B 0,C 180,E1 -10922.91,E2 -10922.91} C_VEL
LIN {X 0,Y 535.928,Z 914.53,A -85,B 0,C 180,E1 -10924.554,E2 -10924.554} C_VEL
LIN {X 0,Y 539.401,Z 894.051,A -85,B 0,C 180,E1 -10925.988,E2 -10925.988} C_VEL
LIN {X 0,Y 542.698,Z 872.602,A -85,B 0,C 180,E1 -10927.256,E2 -10927.256} C_VEL
LIN {X 0,Y 545.604,Z 852.332,A -85,B 0,C 180,E1 -10928.274,E2 -10928.274} C_VEL
LIN {X 0,Y 548.666,Z 827.771,A -85,B 0,C 180,E1 -10929.293,E2 -10929.293} C_VEL
LIN {X 0,Y 550.83,Z 807.489,A -85,B 0,C 180,E1 -10929.969,E2 -10929.969} C_VEL
LIN {X 0,Y 552.99,Z 783.418,A -85,B 0,C 180,E1 -10930.6,E2 -10930.6} C_VEL
LIN {X 0,Y 554.404,Z 759.506,A -85,B 0,C 180,E1 -10931.048,E2 -10931.048} C_VEL
LIN {X 0,Y 561.824,Z 522.16,A -85,B 0,C 180,E1 -10934.435,E2 -10934.435} C_VEL
LIN {X 0,Y 564.354,Z 440.278,A -85,B 0,C 180,E1 -10935.621,E2 -10935.621} C_VEL
LIN {X 0,Y 551.586,Z 418.333,A -85,B 0,C 180,E1 -10937.393,E2 -10937.393} C_VEL
LIN {X 0,Y 539.65,Z 399.517,A -85,B 0,C 180,E1 -10939.152,E2 -10939.152} C_VEL
LIN {X 0,Y 528.463,Z 382.999,A -85,B 0,C 180,E1 -10940.91,E2 -10940.91} C_VEL
LIN {X 0,Y 519.641,Z 370.384,A -85,B 0,C 180,E1 -10942.412,E2 -10942.412} C_VEL
LIN {X 0,Y 516.901,Z 364.587,A -85,B 0,C 180,E1 -10943.568,E2 -10943.568} C_VEL
LIN {X 0,Y 515.368,Z 361.086,A -85,B 0,C 180,E1 -10944.268,E2 -10944.268} C_VEL
LIN {X 0,Y 513.869,Z 357.659,A -85,B 0,C 180,E1 -10944.969,E2 -10944.969} C_VEL
LIN {X 0,Y 513.798,Z 357.158,A -85,B 0,C 180,E1 -10945.1,E2 -10945.1} C_VEL
LIN {X 0,Y 513.75,Z 357.215,A -85,B 0,C 180,E1 -10948.43,E2 -10948.43} C_VEL
LIN {X 0,Y 513.755,Z 357.213,A -85,B 0,C 180,E1 -10951.901,E2 -10951.901} C_VEL
LIN {X 0,Y 513.806,Z 357.213,A -85,B 0,C 180,E1 -10955.266,E2 -10955.266} C_VEL
LIN {X 0,Y 513.752,Z 357.232,A -85,B 0,C 180,E1 -10958.537,E2 -10958.537} C_VEL
LIN {X 0,Y 513.757,Z 357.234,A -85,B 0,C 180,E1 -10962.121,E2 -10962.121} C_VEL
LIN {X 0,Y 513.818,Z 357.221,A -85,B 0,C 180,E1 -10965.461,E2 -10965.461} C_VEL
LIN {X 0,Y 513.759,Z 357.214,A -85,B 0,C 180,E1 -10968.891,E2 -10968.891} C_VEL
LIN {X 0,Y 513.749,Z 357.209,A -85,B 0,C 180,E1 -10972.395,E2 -10972.395} C_VEL
LIN {X 0,Y 513.8,Z 357.224,A -85,B 0,C 180,E1 -10975.759,E2 -10975.759} C_VEL
LIN {X 0,Y 513.764,Z 357.229,A -85,B 0,C 180,E1 -10979.108,E2 -10979.108} C_VEL
LIN {X 0,Y 513.75,Z 357.213,A -85,B 0,C 180,E1 -10982.566,E2 -10982.566} C_VEL
LIN {X 0,Y 513.805,Z 357.21,A -85,B 0,C 180,E1 -10985.92,E2 -10985.92} C_VEL
LIN {X 0,Y 513.767,Z 357.233,A -85,B 0,C 180,E1 -10989.296,E2 -10989.296} C_VEL
LIN {X 0,Y 513.754,Z 357.229,A -85,B 0,C 180,E1 -10992.822,E2 -10992.822} C_VEL
LIN {X 0,Y 513.799,Z 357.208,A -85,B 0,C 180,E1 -10996.158,E2 -10996.158} C_VEL
LIN {X 0,Y 513.775,Z 357.215,A -85,B 0,C 180,E1 -10999.557,E2 -10999.557} C_VEL
LIN {X 0,Y 513.755,Z 357.228,A -85,B 0,C 180,E1 -11002.991,E2 -11002.991} C_VEL
LIN {X 0,Y 513.801,Z 357.229,A -85,B 0,C 180,E1 -11006.341,E2 -11006.341} C_VEL
LIN {X 0,Y 513.77,Z 357.234,A -85,B 0,C 180,E1 -11009.626,E2 -11009.626} C_VEL
LIN {X 0,Y 513.757,Z 357.235,A -85,B 0,C 180,E1 -11013.154,E2 -11013.154} C_VEL
LIN {X 0,Y 513.798,Z 357.224,A -85,B 0,C 180,E1 -11016.548,E2 -11016.548} C_VEL
LIN {X 0,Y 513.803,Z 357.46,A -85,B 0,C 180,E1 -11016.886,E2 -11016.886} C_VEL
LIN {X 0,Y 514.963,Z 360.551,A -85,B 0,C 180,E1 -11017.13,E2 -11017.13} C_VEL
LIN {X 0,Y 517.511,Z 363.048,A -85,B 0,C 180,E1 -11017.56,E2 -11017.56} C_VEL
LIN {X 0,Y 518.326,Z 364.041,A -85,B 0,C 180,E1 -11017.7,E2 -11017.7} C_VEL
LIN {X 0,Y 521.012,Z 367.883,A -85,B 0,C 180,E1 -11018.168,E2 -11018.168} C_VEL
LIN {X 0,Y 522.611,Z 369.697,A -85,B 0,C 180,E1 -11018.431,E2 -11018.431} C_VEL
LIN {X 0,Y 525.859,Z 373.958,A -85,B 0,C 180,E1 -11018.969,E2 -11018.969} C_VEL
LIN {X 0,Y 537.927,Z 389.968,A -85,B 0,C 180,E1 -11020.866,E2 -11020.866} C_VEL
LIN {X 0,Y 548.679,Z 405.342,A -85,B 0,C 180,E1 -11022.451,E2 -11022.451} C_VEL
LIN {X 0,Y 562.382,Z 427.448,A -85,B 0,C 180,E1 -11024.365,E2 -11024.365} C_VEL
LIN {X 0,Y 564.557,Z 431.638,A -85,B 0,C 180,E1 -11024.667,E2 -11024.667} C_VEL
LIN {X 0,Y 556.636,Z 679.871,A -85,B 0,C 180,E1 -11028.206,E2 -11028.206} C_VEL
LIN {X 0,Y 554.512,Z 743.494,A -85,B 0,C 180,E1 -11029.133,E2 -11029.133} C_VEL
LIN {X 0,Y 552.86,Z 768.164,A -85,B 0,C 180,E1 -11029.662,E2 -11029.662} C_VEL
LIN {X 0,Y 550.961,Z 789.727,A -85,B 0,C 180,E1 -11030.276,E2 -11030.276} C_VEL
LIN {X 0,Y 548.369,Z 813.8,A -85,B 0,C 180,E1 -11031.153,E2 -11031.153} C_VEL
LIN {X 0,Y 545.749,Z 834.304,A -85,B 0,C 180,E1 -11032.071,E2 -11032.071} C_VEL
LIN {X 0,Y 542.897,Z 854.394,A -85,B 0,C 180,E1 -11033.128,E2 -11033.128} C_VEL
LIN {X 0,Y 541.111,Z 861.282,A -85,B 0,C 180,E1 -11033.459,E2 -11033.459} C_VEL
LIN {X 0,Y 533.348,Z 878.561,A -85,B 0,C 180,E1 -11034.187,E2 -11034.187} C_VEL
LIN {X 0,Y 531.328,Z 885.016,A -85,B 0,C 180,E1 -11034.595,E2 -11034.595} C_VEL
LIN {X 0,Y 527.704,Z 904.552,A -85,B 0,C 180,E1 -11036.147,E2 -11036.147} C_VEL
LIN {X 0,Y 524.044,Z 923.851,A -85,B 0,C 180,E1 -11037.905,E2 -11037.905} C_VEL
LIN {X 0,Y 520.384,Z 942.006,A -85,B 0,C 180,E1 -11039.844,E2 -11039.844} C_VEL
LIN {X 0,Y 517.142,Z 958.5,A -85,B 0,C 180,E1 -11041.851,E2 -11041.851} C_VEL
LIN {X 0,Y 514.064,Z 973.996,A -85,B 0,C 180,E1 -11044.047,E2 -11044.047} C_VEL
LIN {X 0,Y 511.507,Z 987.663,A -85,B 0,C 180,E1 -11046.254,E2 -11046.254} C_VEL
LIN {X 0,Y 509.201,Z 1000.667,A -85,B 0,C 180,E1 -11048.699,E2 -11048.699} C_VEL
LIN {X 0,Y 507.506,Z 1011.386,A -85,B 0,C 180,E1 -11051.032,E2 -11051.032} C_VEL
LIN {X 0,Y 506.008,Z 1022.224,A -85,B 0,C 180,E1 -11053.822,E2 -11053.822} C_VEL
LIN {X 0,Y 505.141,Z 1029.735,A -85,B 0,C 180,E1 -11056.142,E2 -11056.142} C_VEL
LIN {X 0,Y 504.504,Z 1036.97,A -85,B 0,C 180,E1 -11058.831,E2 -11058.831} C_VEL
LIN {X 0,Y 504.158,Z 1042.311,A -85,B 0,C 180,E1 -11061.446,E2 -11061.446} C_VEL
LIN {X 0,Y 504.011,Z 1046.022,A -85,B 0,C 180,E1 -11063.85,E2 -11063.85} C_VEL
LIN {X 0,Y 503.94,Z 1048.843,A -85,B 0,C 180,E1 -11066.701,E2 -11066.701} C_VEL
LIN {X 0,Y 503.926,Z 1049.877,A -85,B 0,C 180,E1 -11069.091,E2 -11069.091} C_VEL
LIN {X 0,Y 503.924,Z 1049.784,A -85,B 0,C 180,E1 -11071.478,E2 -11071.478} C_VEL
LIN {X 0,Y 503.957,Z 1048.102,A -85,B 0,C 180,E1 -11074.324,E2 -11074.324} C_VEL
LIN {X 0,Y 504.017,Z 1045.363,A -85,B 0,C 180,E1 -11076.722,E2 -11076.722} C_VEL
LIN {X 0,Y 504.224,Z 1041.052,A -85,B 0,C 180,E1 -11079.358,E2 -11079.358} C_VEL
LIN {X 0,Y 504.647,Z 1035.069,A -85,B 0,C 180,E1 -11082.008,E2 -11082.008} C_VEL
LIN {X 0,Y 505.26,Z 1028.618,A -85,B 0,C 180,E1 -11084.322,E2 -11084.322} C_VEL
LIN {X 0,Y 506.412,Z 1019.118,A -85,B 0,C 180,E1 -11087.129,E2 -11087.129} C_VEL
LIN {X 0,Y 507.744,Z 1009.727,A -85,B 0,C 180,E1 -11089.439,E2 -11089.439} C_VEL
LIN {X 0,Y 509.744,Z 997.675,A -85,B 0,C 180,E1 -11092.003,E2 -11092.003} C_VEL
LIN {X 0,Y 512.17,Z 984.032,A -85,B 0,C 180,E1 -11094.449,E2 -11094.449} C_VEL
LIN {X 0,Y 515.036,Z 969.2,A -85,B 0,C 180,E1 -11096.77,E2 -11096.77} C_VEL
LIN {X 0,Y 518.069,Z 953.682,A -85,B 0,C 180,E1 -11098.849,E2 -11098.849} C_VEL
LIN {X 0,Y 521.405,Z 937.174,A -85,B 0,C 180,E1 -11100.799,E2 -11100.799} C_VEL
LIN {X 0,Y 524.98,Z 918.841,A -85,B 0,C 180,E1 -11102.664,E2 -11102.664} C_VEL
LIN {X 0,Y 528.292,Z 901.547,A -85,B 0,C 180,E1 -11104.203,E2 -11104.203} C_VEL
LIN {X 0,Y 532.287,Z 879.616,A -85,B 0,C 180,E1 -11105.88,E2 -11105.88} C_VEL
LIN {X 0,Y 535.416,Z 860.982,A -85,B 0,C 180,E1 -11107.1,E2 -11107.1} C_VEL
LIN {X 0,Y 538.917,Z 838.375,A -85,B 0,C 180,E1 -11108.362,E2 -11108.362} C_VEL
LIN {X 0,Y 541.693,Z 817.69,A -85,B 0,C 180,E1 -11109.319,E2 -11109.319} C_VEL
LIN {X 0,Y 544.164,Z 796.818,A -85,B 0,C 180,E1 -11110.128,E2 -11110.128} C_VEL
LIN {X 0,Y 546.501,Z 772.352,A -85,B 0,C 180,E1 -11110.872,E2 -11110.872} C_VEL
LIN {X 0,Y 548.045,Z 751.688,A -85,B 0,C 180,E1 -11111.352,E2 -11111.352} C_VEL
LIN {X 0,Y 549.375,Z 723.105,A -85,B 0,C 180,E1 -11111.829,E2 -11111.829} C_VEL
LIN {X 0,Y 557.744,Z 468.891,A -85,B 0,C 180,E1 -11115.476,E2 -11115.476} C_VEL
LIN {X 0,Y 558.764,Z 434.451,A -85,B 0,C 180,E1 -11115.992,E2 -11115.992} C_VEL
LIN {X 0,Y 547.25,Z 415.386,A -85,B 0,C 180,E1 -11117.625,E2 -11117.625} C_VEL
LIN {X 0,Y 537.124,Z 400.381,A -85,B 0,C 180,E1 -11119.13,E2 -11119.13} C_VEL
LIN {X 0,Y 525.488,Z 384.617,A -85,B 0,C 180,E1 -11120.963,E2 -11120.963} C_VEL
LIN {X 0,Y 521.74,Z 379.819,A -85,B 0,C 180,E1 -11121.581,E2 -11121.581} C_VEL
LIN {X 0,Y 517.784,Z 374.653,A -85,B 0,C 180,E1 -11122.254,E2 -11122.254} C_VEL
LIN {X 0,Y 514.026,Z 369.74,A -85,B 0,C 180,E1 -11122.914,E2 -11122.914} C_VEL
LIN {X 0,Y 511.082,Z 366.286,A -85,B 0,C 180,E1 -11123.435,E2 -11123.435} C_VEL
LIN {X 0,Y 509.813,Z 364.154,A -85,B 0,C 180,E1 -11123.679,E2 -11123.679} C_VEL
LIN {X 0,Y 507.125,Z 361.685,A -85,B 0,C 180,E1 -11124.155,E2 -11124.155} C_VEL
LIN {X 0,Y 505.887,Z 358.671,A -85,B 0,C 180,E1 -11124.423,E2 -11124.423} C_VEL
LIN {X 0,Y 505.816,Z 358.224,A -85,B 0,C 180,E1 -11124.467,E2 -11124.467} C_VEL
LIN {X 0,Y 505.866,Z 358.212,A -85,B 0,C 180,E1 -11127.879,E2 -11127.879} C_VEL
LIN {X 0,Y 505.818,Z 358.221,A -85,B 0,C 180,E1 -11131.162,E2 -11131.162} C_VEL
LIN {X 0,Y 505.813,Z 358.224,A -85,B 0,C 180,E1 -11134.723,E2 -11134.723} C_VEL
LIN {X 0,Y 505.868,Z 358.219,A -85,B 0,C 180,E1 -11138.064,E2 -11138.064} C_VEL
LIN {X 0,Y 505.824,Z 358.211,A -85,B 0,C 180,E1 -11141.442,E2 -11141.442} C_VEL
LIN {X 0,Y 505.809,Z 358.2,A -85,B 0,C 180,E1 -11144.874,E2 -11144.874} C_VEL
LIN {X 0,Y 505.857,Z 358.199,A -85,B 0,C 180,E1 -11148.253,E2 -11148.253} C_VEL
LIN {X 0,Y 505.83,Z 358.225,A -85,B 0,C 180,E1 -11151.703,E2 -11151.703} C_VEL
LIN {X 0,Y 505.809,Z 358.217,A -85,B 0,C 180,E1 -11155.124,E2 -11155.124} C_VEL
LIN {X 0,Y 505.85,Z 358.194,A -85,B 0,C 180,E1 -11158.528,E2 -11158.528} C_VEL
LIN {X 0,Y 505.824,Z 358.211,A -85,B 0,C 180,E1 -11161.812,E2 -11161.812} C_VEL
LIN {X 0,Y 505.809,Z 358.224,A -85,B 0,C 180,E1 -11165.331,E2 -11165.331} C_VEL
LIN {X 0,Y 505.858,Z 358.2,A -85,B 0,C 180,E1 -11168.64,E2 -11168.64} C_VEL
LIN {X 0,Y 505.831,Z 358.198,A -85,B 0,C 180,E1 -11172.095,E2 -11172.095} C_VEL
LIN {X 0,Y 505.808,Z 358.214,A -85,B 0,C 180,E1 -11175.478,E2 -11175.478} C_VEL
LIN {X 0,Y 505.847,Z 358.217,A -85,B 0,C 180,E1 -11178.916,E2 -11178.916} C_VEL
LIN {X 0,Y 505.839,Z 358.217,A -85,B 0,C 180,E1 -11182.317,E2 -11182.317} C_VEL
LIN {X 0,Y 505.809,Z 358.219,A -85,B 0,C 180,E1 -11185.779,E2 -11185.779} C_VEL
LIN {X 0,Y 505.834,Z 358.216,A -85,B 0,C 180,E1 -11189.226,E2 -11189.226} C_VEL
LIN {X 0,Y 505.841,Z 358.218,A -85,B 0,C 180,E1 -11192.525,E2 -11192.525} C_VEL
LIN {X 0,Y 505.826,Z 358.356,A -85,B 0,C 180,E1 -11193.838,E2 -11193.838} C_VEL
LIN {X 0,Y 507.295,Z 361.901,A -85,B 0,C 180,E1 -11194.587,E2 -11194.587} C_VEL
LIN {X 0,Y 508.091,Z 363.478,A -85,B 0,C 180,E1 -11194.937,E2 -11194.937} C_VEL
LIN {X 0,Y 511.474,Z 370.578,A -85,B 0,C 180,E1 -11196.393,E2 -11196.393} C_VEL
LIN {X 0,Y 523.138,Z 387.001,A -85,B 0,C 180,E1 -11198.438,E2 -11198.438} C_VEL
LIN {X 0,Y 532.536,Z 400.734,A -85,B 0,C 180,E1 -11199.969,E2 -11199.969} C_VEL
LIN {X 0,Y 544.584,Z 419.544,A -85,B 0,C 180,E1 -11201.815,E2 -11201.815} C_VEL
LIN {X 0,Y 557.053,Z 440.663,A -85,B 0,C 180,E1 -11203.608,E2 -11203.608} C_VEL
LIN {X 0,Y 558.816,Z 444.201,A -85,B 0,C 180,E1 -11203.86,E2 -11203.86} C_VEL
LIN {X 0,Y 550.463,Z 697.131,A -85,B 0,C 180,E1 -11207.495,E2 -11207.495} C_VEL
LIN {X 0,Y 548.133,Z 765.248,A -85,B 0,C 180,E1 -11208.493,E2 -11208.493} C_VEL
LIN {X 0,Y 546.267,Z 790.565,A -85,B 0,C 180,E1 -11209.024,E2 -11209.024} C_VEL
LIN {X 0,Y 544.172,Z 812.301,A -85,B 0,C 180,E1 -11209.634,E2 -11209.634} C_VEL
LIN {X 0,Y 541.221,Z 837.327,A -85,B 0,C 180,E1 -11210.541,E2 -11210.541} C_VEL
LIN {X 0,Y 538.44,Z 857.889,A -85,B 0,C 180,E1 -11211.462,E2 -11211.462} C_VEL
LIN {X 0,Y 534.858,Z 881.339,A -85,B 0,C 180,E1 -11212.721,E2 -11212.721} C_VEL
LIN {X 0,Y 531.554,Z 901.109,A -85,B 0,C 180,E1 -11213.985,E2 -11213.985} C_VEL
LIN {X 0,Y 527.781,Z 922.37,A -85,B 0,C 180,E1 -11215.562,E2 -11215.562} C_VEL
LIN {X 0,Y 524.205,Z 941.212,A -85,B 0,C 180,E1 -11217.2,E2 -11217.2} C_VEL
LIN {X 0,Y 520.601,Z 960.189,A -85,B 0,C 180,E1 -11219.084,E2 -11219.084} C_VEL
LIN {X 0,Y 517.234,Z 977.552,A -85,B 0,C 180,E1 -11221.1,E2 -11221.1} C_VEL
LIN {X 0,Y 514.258,Z 993.421,A -85,B 0,C 180,E1 -11223.187,E2 -11223.187} C_VEL
LIN {X 0,Y 511.492,Z 1008.647,A -85,B 0,C 180,E1 -11225.517,E2 -11225.517} C_VEL
LIN {X 0,Y 509.352,Z 1021.369,A -85,B 0,C 180,E1 -11227.736,E2 -11227.736} C_VEL
LIN {X 0,Y 507.384,Z 1034.393,A -85,B 0,C 180,E1 -11230.388,E2 -11230.388} C_VEL
LIN {X 0,Y 506.145,Z 1043.916,A -85,B 0,C 180,E1 -11232.644,E2 -11232.644} C_VEL
LIN {X 0,Y 505.059,Z 1054.051,A -85,B 0,C 180,E1 -11235.49,E2 -11235.49} C_VEL
LIN {X 0,Y 504.486,Z 1060.989,A -85,B 0,C 180,E1 -11237.872,E2 -11237.872} C_VEL
LIN {X 0,Y 504.125,Z 1067.297,A -85,B 0,C 180,E1 -11240.525,E2 -11240.525} C_VEL
LIN {X 0,Y 503.962,Z 1071.857,A -85,B 0,C 180,E1 -11243.163,E2 -11243.163} C_VEL
LIN {X 0,Y 503.928,Z 1074.65,A -85,B 0,C 180,E1 -11245.448,E2 -11245.448} C_VEL
LIN {X 0,Y 503.919,Z 1076.555,A -85,B 0,C 180,E1 -11248.067,E2 -11248.067} C_VEL
LIN {X 0,Y 503.918,Z 1076.828,A -85,B 0,C 180,E1 -11250.682,E2 -11250.682} C_VEL
LIN {X 0,Y 503.927,Z 1075.933,A -85,B 0,C 180,E1 -11252.957,E2 -11252.957} C_VEL
LIN {X 0,Y 503.941,Z 1073.606,A -85,B 0,C 180,E1 -11255.579,E2 -11255.579} C_VEL
LIN {X 0,Y 504.042,Z 1069.421,A -85,B 0,C 180,E1 -11258.326,E2 -11258.326} C_VEL
LIN {X 0,Y 504.268,Z 1064.452,A -85,B 0,C 180,E1 -11260.742,E2 -11260.742} C_VEL
LIN {X 0,Y 504.815,Z 1056.76,A -85,B 0,C 180,E1 -11263.633,E2 -11263.633} C_VEL
LIN {X 0,Y 505.567,Z 1048.932,A -85,B 0,C 180,E1 -11266.013,E2 -11266.013} C_VEL
LIN {X 0,Y 506.813,Z 1038.736,A -85,B 0,C 180,E1 -11268.639,E2 -11268.639} C_VEL
LIN {X 0,Y 508.409,Z 1027.347,A -85,B 0,C 180,E1 -11271.094,E2 -11271.094} C_VEL
LIN {X 0,Y 510.574,Z 1014.122,A -85,B 0,C 180,E1 -11273.578,E2 -11273.578} C_VEL
LIN {X 0,Y 513.08,Z 999.701,A -85,B 0,C 180,E1 -11275.883,E2 -11275.883} C_VEL
LIN {X 0,Y 516.016,Z 984.005,A -85,B 0,C 180,E1 -11278.09,E2 -11278.09} C_VEL
LIN {X 0,Y 519.289,Z 966.81,A -85,B 0,C 180,E1 -11280.169,E2 -11280.169} C_VEL
LIN {X 0,Y 522.468,Z 950.352,A -85,B 0,C 180,E1 -11281.921,E2 -11281.921} C_VEL
LIN {X 0,Y 526.355,Z 929.712,A -85,B 0,C 180,E1 -11283.821,E2 -11283.821} C_VEL
LIN {X 0,Y 529.719,Z 911.348,A -85,B 0,C 180,E1 -11285.282,E2 -11285.282} C_VEL
LIN {X 0,Y 533.671,Z 888.505,A -85,B 0,C 180,E1 -11286.838,E2 -11286.838} C_VEL
LIN {X 0,Y 536.692,Z 869.498,A -85,B 0,C 180,E1 -11287.938,E2 -11287.938} C_VEL
LIN {X 0,Y 540.084,Z 846.231,A -85,B 0,C 180,E1 -11289.079,E2 -11289.079} C_VEL
LIN {X 0,Y 542.772,Z 824.576,A -85,B 0,C 180,E1 -11289.941,E2 -11289.941} C_VEL
LIN {X 0,Y 545.052,Z 803.732,A -85,B 0,C 180,E1 -11290.62,E2 -11290.62} C_VEL
LIN {X 0,Y 547.225,Z 778.356,A -85,B 0,C 180,E1 -11291.249,E2 -11291.249} C_VEL
LIN {X 0,Y 548.516,Z 756.139,A -85,B 0,C 180,E1 -11291.649,E2 -11291.649} C_VEL
LIN {X 0,Y 556.607,Z 507.561,A -85,B 0,C 180,E1 -11295.22,E2 -11295.22} C_VEL
LIN {X 0,Y 558.653,Z 443.531,A -85,B 0,C 180,E1 -11296.159,E2 -11296.159} C_VEL
LIN {X 0,Y 546.051,Z 422.037,A -85,B 0,C 180,E1 -11297.953,E2 -11297.953} C_VEL
LIN {X 0,Y 533.677,Z 402.369,A -85,B 0,C 180,E1 -11299.835,E2 -11299.835} C_VEL
LIN {X 0,Y 520.475,Z 383.07,A -85,B 0,C 180,E1 -11301.996,E2 -11301.996} C_VEL
LIN {X 0,Y 514.132,Z 374.489,A -85,B 0,C 180,E1 -11303.097,E2 -11303.097} C_VEL
LIN {X 0,Y 511.16,Z 370.112,A -85,B 0,C 180,E1 -11303.651,E2 -11303.651} C_VEL
LIN {X 0,Y 507.577,Z 362.207,A -85,B 0,C 180,E1 -11305.298,E2 -11305.298} C_VEL
LIN {X 0,Y 505.983,Z 359.124,A -85,B 0,C 180,E1 -11305.996,E2 -11305.996} C_VEL
LIN {X 0,Y 505.805,Z 358.179,A -85,B 0,C 180,E1 -11306.202,E2 -11306.202} C_VEL
LIN {X 0,Y 505.837,Z 358.202,A -85,B 0,C 180,E1 -11309.6,E2 -11309.6} C_VEL
LIN {X 0,Y 505.849,Z 358.2,A -85,B 0,C 180,E1 -11312.959,E2 -11312.959} C_VEL
LIN {X 0,Y 505.81,Z 358.205,A -85,B 0,C 180,E1 -11316.341,E2 -11316.341} C_VEL
LIN {X 0,Y 505.837,Z 358.2,A -85,B 0,C 180,E1 -11319.762,E2 -11319.762} C_VEL
LIN {X 0,Y 505.847,Z 358.204,A -85,B 0,C 180,E1 -11323.108,E2 -11323.108} C_VEL
LIN {X 0,Y 505.812,Z 358.222,A -85,B 0,C 180,E1 -11326.511,E2 -11326.511} C_VEL
LIN {X 0,Y 505.834,Z 358.219,A -85,B 0,C 180,E1 -11329.982,E2 -11329.982} C_VEL
LIN {X 0,Y 505.849,Z 358.194,A -85,B 0,C 180,E1 -11333.303,E2 -11333.303} C_VEL
LIN {X 0,Y 505.81,Z 358.204,A -85,B 0,C 180,E1 -11336.714,E2 -11336.714} C_VEL
LIN {X 0,Y 505.83,Z 358.219,A -85,B 0,C 180,E1 -11340.227,E2 -11340.227} C_VEL
LIN {X 0,Y 505.86,Z 358.21,A -85,B 0,C 180,E1 -11343.626,E2 -11343.626} C_VEL
LIN {X 0,Y 505.812,Z 358.197,A -85,B 0,C 180,E1 -11347.04,E2 -11347.04} C_VEL
LIN {X 0,Y 505.818,Z 358.204,A -85,B 0,C 180,E1 -11350.594,E2 -11350.594} C_VEL
LIN {X 0,Y 505.872,Z 358.216,A -85,B 0,C 180,E1 -11354.071,E2 -11354.071} C_VEL
LIN {X 0,Y 505.834,Z 358.218,A -85,B 0,C 180,E1 -11357.485,E2 -11357.485} C_VEL
LIN {X 0,Y 505.815,Z 358.209,A -85,B 0,C 180,E1 -11360.965,E2 -11360.965} C_VEL
LIN {X 0,Y 505.857,Z 358.199,A -85,B 0,C 180,E1 -11364.325,E2 -11364.325} C_VEL
LIN {X 0,Y 505.834,Z 358.202,A -85,B 0,C 180,E1 -11367.68,E2 -11367.68} C_VEL
LIN {X 0,Y 505.816,Z 358.204,A -85,B 0,C 180,E1 -11371.136,E2 -11371.136} C_VEL
LIN {X 0,Y 505.853,Z 358.201,A -85,B 0,C 180,E1 -11374.562,E2 -11374.562} C_VEL
LIN {X 0,Y 505.844,Z 358.345,A -85,B 0,C 180,E1 -11375.679,E2 -11375.679} C_VEL
LIN {X 0,Y 506.958,Z 361.401,A -85,B 0,C 180,E1 -11375.928,E2 -11375.928} C_VEL
LIN {X 0,Y 509.631,Z 364.05,A -85,B 0,C 180,E1 -11376.406,E2 -11376.406} C_VEL
LIN {X 0,Y 510.423,Z 365.016,A -85,B 0,C 180,E1 -11376.55,E2 -11376.55} C_VEL
LIN {X 0,Y 513.027,Z 368.834,A -85,B 0,C 180,E1 -11377.031,E2 -11377.031} C_VEL
LIN {X 0,Y 515.004,Z 370.914,A -85,B 0,C 180,E1 -11377.371,E2 -11377.371} C_VEL
LIN {X 0,Y 518.314,Z 375.17,A -85,B 0,C 180,E1 -11377.945,E2 -11377.945} C_VEL
LIN {X 0,Y 522.704,Z 380.838,A -85,B 0,C 180,E1 -11378.686,E2 -11378.686} C_VEL
LIN {X 0,Y 535.167,Z 397.795,A -85,B 0,C 180,E1 -11380.68,E2 -11380.68} C_VEL
LIN {X 0,Y 544.471,Z 411.112,A -85,B 0,C 180,E1 -11382.073,E2 -11382.073} C_VEL
LIN {X 0,Y 557.963,Z 433.086,A -85,B 0,C 180,E1 -11383.999,E2 -11383.999} C_VEL
LIN {X 0,Y 558.85,Z 435.059,A -85,B 0,C 180,E1 -11384.129,E2 -11384.129} C_VEL
LIN {X 0,Y 550.578,Z 683.773,A -85,B 0,C 180,E1 -11387.704,E2 -11387.704} C_VEL
LIN {X 0,Y 548.471,Z 744.053,A -85,B 0,C 180,E1 -11388.591,E2 -11388.591} C_VEL
LIN {X 0,Y 546.752,Z 768.653,A -85,B 0,C 180,E1 -11389.125,E2 -11389.125} C_VEL
LIN {X 0,Y 544.768,Z 790.386,A -85,B 0,C 180,E1 -11389.749,E2 -11389.749} C_VEL
LIN {X 0,Y 542.118,Z 814.024,A -85,B 0,C 180,E1 -11390.619,E2 -11390.619} C_VEL
LIN {X 0,Y 539.405,Z 834.528,A -85,B 0,C 180,E1 -11391.544,E2 -11391.544} C_VEL
LIN {X 0,Y 536.212,Z 856.123,A -85,B 0,C 180,E1 -11392.697,E2 -11392.697} C_VEL
LIN {X 0,Y 532.743,Z 876.836,A -85,B 0,C 180,E1 -11394.023,E2 -11394.023} C_VEL
LIN {X 0,Y 531.328,Z 885.016,A -85,B 0,C 180,E1 -11394.595,E2 -11394.595} C_VEL
LIN {X 0,Y 529.316,Z 891.434,A -85,B 0,C 180,E1 -11395.02,E2 -11395.02} C_VEL
LIN {X 0,Y 521.271,Z 907.731,A -85,B 0,C 180,E1 -11395.96,E2 -11395.96} C_VEL
LIN {X 0,Y 519.189,Z 913.758,A -85,B 0,C 180,E1 -11396.442,E2 -11396.442} C_VEL
LIN {X 0,Y 515.661,Z 930.925,A -85,B 0,C 180,E1 -11398.136,E2 -11398.136} C_VEL
LIN {X 0,Y 512.013,Z 948.642,A -85,B 0,C 180,E1 -11400.134,E2 -11400.134} C_VEL
LIN {X 0,Y 508.651,Z 964.616,A -85,B 0,C 180,E1 -11402.232,E2 -11402.232} C_VEL
LIN {X 0,Y 505.651,Z 979.55,A -85,B 0,C 180,E1 -11404.464,E2 -11404.464} C_VEL
LIN {X 0,Y 503,Z 993.036,A -85,B 0,C 180,E1 -11406.822,E2 -11406.822} C_VEL
LIN {X 0,Y 500.878,Z 1004.848,A -85,B 0,C 180,E1 -11409.186,E2 -11409.186} C_VEL
LIN {X 0,Y 499.02,Z 1016.356,A -85,B 0,C 180,E1 -11411.906,E2 -11411.906} C_VEL
LIN {X 0,Y 497.807,Z 1025.234,A -85,B 0,C 180,E1 -11414.386,E2 -11414.386} C_VEL
LIN {X 0,Y 496.844,Z 1033.86,A -85,B 0,C 180,E1 -11417.329,E2 -11417.329} C_VEL
LIN {X 0,Y 496.351,Z 1039.619,A -85,B 0,C 180,E1 -11419.789,E2 -11419.789} C_VEL
LIN {X 0,Y 496.083,Z 1044.683,A -85,B 0,C 180,E1 -11422.598,E2 -11422.598} C_VEL
LIN {X 0,Y 495.966,Z 1047.781,A -85,B 0,C 180,E1 -11425.143,E2 -11425.143} C_VEL
LIN {X 0,Y 495.931,Z 1049.591,A -85,B 0,C 180,E1 -11427.573,E2 -11427.573} C_VEL
LIN {X 0,Y 495.921,Z 1050.198,A -85,B 0,C 180,E1 -11430.462,E2 -11430.462} C_VEL
LIN {X 0,Y 495.933,Z 1049.376,A -85,B 0,C 180,E1 -11432.889,E2 -11432.889} C_VEL
LIN {X 0,Y 495.974,Z 1047.424,A -85,B 0,C 180,E1 -11435.321,E2 -11435.321} C_VEL
LIN {X 0,Y 496.124,Z 1043.497,A -85,B 0,C 180,E1 -11438.227,E2 -11438.227} C_VEL
LIN {X 0,Y 496.419,Z 1038.814,A -85,B 0,C 180,E1 -11440.679,E2 -11440.679} C_VEL
LIN {X 0,Y 497.048,Z 1031.962,A -85,B 0,C 180,E1 -11443.495,E2 -11443.495} C_VEL
LIN {X 0,Y 497.973,Z 1023.945,A -85,B 0,C 180,E1 -11446.087,E2 -11446.087} C_VEL
LIN {X 0,Y 499.354,Z 1014.327,A -85,B 0,C 180,E1 -11448.715,E2 -11448.715} C_VEL
LIN {X 0,Y 501.192,Z 1002.956,A -85,B 0,C 180,E1 -11451.301,E2 -11451.301} C_VEL
LIN {X 0,Y 503.403,Z 990.996,A -85,B 0,C 180,E1 -11453.655,E2 -11453.655} C_VEL
LIN {X 0,Y 506.274,Z 976.309,A -85,B 0,C 180,E1 -11456.131,E2 -11456.131} C_VEL
LIN {X 0,Y 509.242,Z 961.888,A -85,B 0,C 180,E1 -11458.242,E2 -11458.242} C_VEL
LIN {X 0,Y 512.957,Z 944.003,A -85,B 0,C 180,E1 -11460.505,E2 -11460.505} C_VEL
LIN {X 0,Y 516.268,Z 928.146,A -85,B 0,C 180,E1 -11462.248,E2 -11462.248} C_VEL
LIN {X 0,Y 520.411,Z 907.724,A -85,B 0,C 180,E1 -11464.194,E2 -11464.194} C_VEL
LIN {X 0,Y 523.861,Z 889.827,A -85,B 0,C 180,E1 -11465.661,E2 -11465.661} C_VEL
LIN {X 0,Y 527.61,Z 869.374,A -85,B 0,C 180,E1 -11467.119,E2 -11467.119} C_VEL
LIN {X 0,Y 530.958,Z 848.836,A -85,B 0,C 180,E1 -11468.353,E2 -11468.353} C_VEL
LIN {X 0,Y 534.236,Z 827.332,A -85,B 0,C 180,E1 -11469.451,E2 -11469.451} C_VEL
LIN {X 0,Y 537.196,Z 804.049,A -85,B 0,C 180,E1 -11470.423,E2 -11470.423} C_VEL
LIN {X 0,Y 539.536,Z 782.514,A -85,B 0,C 180,E1 -11471.15,E2 -11471.15} C_VEL
LIN {X 0,Y 541.692,Z 757.229,A -85,B 0,C 180,E1 -11471.8,E2 -11471.8} C_VEL
LIN {X 0,Y 542.946,Z 735.564,A -85,B 0,C 180,E1 -11472.205,E2 -11472.205} C_VEL
LIN {X 0,Y 551.514,Z 487.038,A -85,B 0,C 180,E1 -11475.808,E2 -11475.808} C_VEL
LIN {X 0,Y 553.122,Z 437.841,A -85,B 0,C 180,E1 -11476.541,E2 -11476.541} C_VEL
LIN {X 0,Y 539.633,Z 415.831,A -85,B 0,C 180,E1 -11478.515,E2 -11478.515} C_VEL
LIN {X 0,Y 526.646,Z 397.302,A -85,B 0,C 180,E1 -11480.538,E2 -11480.538} C_VEL
LIN {X 0,Y 518.055,Z 386.068,A -85,B 0,C 180,E1 -11481.962,E2 -11481.962} C_VEL
LIN {X 0,Y 514,Z 380.79,A -85,B 0,C 180,E1 -11482.666,E2 -11482.666} C_VEL
LIN {X 0,Y 510.407,Z 376.156,A -85,B 0,C 180,E1 -11483.309,E2 -11483.309} C_VEL
LIN {X 0,Y 507.203,Z 371.948,A -85,B 0,C 180,E1 -11483.9,E2 -11483.9} C_VEL
LIN {X 0,Y 505.683,Z 370.313,A -85,B 0,C 180,E1 -11484.177,E2 -11484.177} C_VEL
LIN {X 0,Y 502.928,Z 366.731,A -85,B 0,C 180,E1 -11484.704,E2 -11484.704} C_VEL
LIN {X 0,Y 502.136,Z 365.321,A -85,B 0,C 180,E1 -11484.867,E2 -11484.867} C_VEL
LIN {X 0,Y 499.431,Z 362.995,A -85,B 0,C 180,E1 -11485.371,E2 -11485.371} C_VEL
LIN {X 0,Y 498.04,Z 359.884,A -85,B 0,C 180,E1 -11485.683,E2 -11485.683} C_VEL
LIN {X 0,Y 497.923,Z 359.19,A -85,B 0,C 180,E1 -11485.743,E2 -11485.743} C_VEL
LIN {X 0,Y 497.88,Z 359.194,A -85,B 0,C 180,E1 -11489.195,E2 -11489.195} C_VEL
LIN {X 0,Y 497.872,Z 359.192,A -85,B 0,C 180,E1 -11492.748,E2 -11492.748} C_VEL
LIN {X 0,Y 497.909,Z 359.187,A -85,B 0,C 180,E1 -11496.194,E2 -11496.194} C_VEL
LIN {X 0,Y 497.883,Z 359.197,A -85,B 0,C 180,E1 -11499.424,E2 -11499.424} C_VEL
LIN {X 0,Y 497.871,Z 359.213,A -85,B 0,C 180,E1 -11502.949,E2 -11502.949} C_VEL
LIN {X 0,Y 497.906,Z 359.209,A -85,B 0,C 180,E1 -11506.411,E2 -11506.411} C_VEL
LIN {X 0,Y 497.911,Z 359.187,A -85,B 0,C 180,E1 -11509.938,E2 -11509.938} C_VEL
LIN {X 0,Y 497.867,Z 359.19,A -85,B 0,C 180,E1 -11513.311,E2 -11513.311} C_VEL
LIN {X 0,Y 497.888,Z 359.207,A -85,B 0,C 180,E1 -11516.776,E2 -11516.776} C_VEL
LIN {X 0,Y 497.933,Z 359.201,A -85,B 0,C 180,E1 -11520.23,E2 -11520.23} C_VEL
LIN {X 0,Y 497.875,Z 359.186,A -85,B 0,C 180,E1 -11523.685,E2 -11523.685} C_VEL
LIN {X 0,Y 497.868,Z 359.19,A -85,B 0,C 180,E1 -11527.269,E2 -11527.269} C_VEL
LIN {X 0,Y 497.917,Z 359.203,A -85,B 0,C 180,E1 -11530.647,E2 -11530.647} C_VEL
LIN {X 0,Y 497.891,Z 359.207,A -85,B 0,C 180,E1 -11534.073,E2 -11534.073} C_VEL
LIN {X 0,Y 497.868,Z 359.196,A -85,B 0,C 180,E1 -11537.533,E2 -11537.533} C_VEL
LIN {X 0,Y 497.907,Z 359.185,A -85,B 0,C 180,E1 -11540.964,E2 -11540.964} C_VEL
LIN {X 0,Y 497.889,Z 359.19,A -85,B 0,C 180,E1 -11544.252,E2 -11544.252} C_VEL
LIN {X 0,Y 497.872,Z 359.196,A -85,B 0,C 180,E1 -11547.666,E2 -11547.666} C_VEL
LIN {X 0,Y 497.912,Z 359.193,A -85,B 0,C 180,E1 -11551.071,E2 -11551.071} C_VEL
LIN {X 0,Y 497.93,Z 359.322,A -85,B 0,C 180,E1 -11552.663,E2 -11552.663} C_VEL
LIN {X 0,Y 499.268,Z 362.801,A -85,B 0,C 180,E1 -11553.418,E2 -11553.418} C_VEL
LIN {X 0,Y 500.274,Z 364.86,A -85,B 0,C 180,E1 -11553.892,E2 -11553.892} C_VEL
LIN {X 0,Y 502.324,Z 369.085,A -85,B 0,C 180,E1 -11554.84,E2 -11554.84} C_VEL
LIN {X 0,Y 503.238,Z 370.811,A -85,B 0,C 180,E1 -11555.115,E2 -11555.115} C_VEL
LIN {X 0,Y 509.567,Z 379.333,A -85,B 0,C 180,E1 -11556.307,E2 -11556.307} C_VEL
LIN {X 0,Y 518.631,Z 391.928,A -85,B 0,C 180,E1 -11557.918,E2 -11557.918} C_VEL
LIN {X 0,Y 530.499,Z 409.549,A -85,B 0,C 180,E1 -11559.89,E2 -11559.89} C_VEL
LIN {X 0,Y 542.703,Z 429.138,A -85,B 0,C 180,E1 -11561.78,E2 -11561.78} C_VEL
LIN {X 0,Y 553.157,Z 447.315,A -85,B 0,C 180,E1 -11563.308,E2 -11563.308} C_VEL
LIN {X 0,Y 544.497,Z 699.121,A -85,B 0,C 180,E1 -11566.955,E2 -11566.955} C_VEL
LIN {X 0,Y 542.141,Z 765.159,A -85,B 0,C 180,E1 -11567.932,E2 -11567.932} C_VEL
LIN {X 0,Y 540.222,Z 790.362,A -85,B 0,C 180,E1 -11568.465,E2 -11568.465} C_VEL
LIN {X 0,Y 538.076,Z 811.91,A -85,B 0,C 180,E1 -11569.073,E2 -11569.073} C_VEL
LIN {X 0,Y 534.993,Z 837.118,A -85,B 0,C 180,E1 -11569.989,E2 -11569.989} C_VEL
LIN {X 0,Y 532.108,Z 857.677,A -85,B 0,C 180,E1 -11570.917,E2 -11570.917} C_VEL
LIN {X 0,Y 528.382,Z 881.126,A -85,B 0,C 180,E1 -11572.184,E2 -11572.184} C_VEL
LIN {X 0,Y 524.92,Z 901.034,A -85,B 0,C 180,E1 -11573.469,E2 -11573.469} C_VEL
LIN {X 0,Y 521.101,Z 921.767,A -85,B 0,C 180,E1 -11575.018,E2 -11575.018} C_VEL
LIN {X 0,Y 517.296,Z 940.995,A -85,B 0,C 180,E1 -11576.705,E2 -11576.705} C_VEL
LIN {X 0,Y 513.519,Z 959.971,A -85,B 0,C 180,E1 -11578.61,E2 -11578.61} C_VEL
LIN {X 0,Y 509.991,Z 977.333,A -85,B 0,C 180,E1 -11580.649,E2 -11580.649} C_VEL
LIN {X 0,Y 506.711,Z 994.04,A -85,B 0,C 180,E1 -11582.881,E2 -11582.881} C_VEL
LIN {X 0,Y 503.822,Z 1009.136,A -85,B 0,C 180,E1 -11585.244,E2 -11585.244} C_VEL
LIN {X 0,Y 501.389,Z 1023.061,A -85,B 0,C 180,E1 -11587.734,E2 -11587.734} C_VEL
LIN {X 0,Y 499.508,Z 1034.862,A -85,B 0,C 180,E1 -11590.227,E2 -11590.227} C_VEL
LIN {X 0,Y 498.128,Z 1045.094,A -85,B 0,C 180,E1 -11592.718,E2 -11592.718} C_VEL
LIN {X 0,Y 497.08,Z 1054.392,A -85,B 0,C 180,E1 -11595.437,E2 -11595.437} C_VEL
LIN {X 0,Y 496.502,Z 1061.08,A -85,B 0,C 180,E1 -11597.792,E2 -11597.792} C_VEL
LIN {X 0,Y 496.114,Z 1067.522,A -85,B 0,C 180,E1 -11600.604,E2 -11600.604} C_VEL
LIN {X 0,Y 495.962,Z 1071.805,A -85,B 0,C 180,E1 -11603.169,E2 -11603.169} C_VEL
LIN {X 0,Y 495.928,Z 1074.552,A -85,B 0,C 180,E1 -11605.49,E2 -11605.49} C_VEL
LIN {X 0,Y 495.917,Z 1076.405,A -85,B 0,C 180,E1 -11608.267,E2 -11608.267} C_VEL
LIN {X 0,Y 495.924,Z 1076.592,A -85,B 0,C 180,E1 -11610.809,E2 -11610.809} C_VEL
LIN {X 0,Y 495.931,Z 1075.65,A -85,B 0,C 180,E1 -11613.12,E2 -11613.12} C_VEL
LIN {X 0,Y 495.949,Z 1073.104,A -85,B 0,C 180,E1 -11615.902,E2 -11615.902} C_VEL
LIN {X 0,Y 496.052,Z 1068.995,A -85,B 0,C 180,E1 -11618.578,E2 -11618.578} C_VEL
LIN {X 0,Y 496.308,Z 1063.975,A -85,B 0,C 180,E1 -11621.034,E2 -11621.034} C_VEL
LIN {X 0,Y 496.908,Z 1056.182,A -85,B 0,C 180,E1 -11623.973,E2 -11623.973} C_VEL
LIN {X 0,Y 497.703,Z 1048.499,A -85,B 0,C 180,E1 -11626.335,E2 -11626.335} C_VEL
LIN {X 0,Y 499.067,Z 1037.993,A -85,B 0,C 180,E1 -11629.061,E2 -11629.061} C_VEL
LIN {X 0,Y 500.743,Z 1026.885,A -85,B 0,C 180,E1 -11631.484,E2 -11631.484} C_VEL
LIN {X 0,Y 502.952,Z 1014.064,A -85,B 0,C 180,E1 -11633.926,E2 -11633.926} C_VEL
LIN {X 0,Y 505.627,Z 999.477,A -85,B 0,C 180,E1 -11636.293,E2 -11636.293} C_VEL
LIN {X 0,Y 508.533,Z 984.636,A -85,B 0,C 180,E1 -11638.413,E2 -11638.413} C_VEL
LIN {X 0,Y 511.986,Z 967.403,A -85,B 0,C 180,E1 -11640.542,E2 -11640.542} C_VEL
LIN {X 0,Y 515.303,Z 950.944,A -85,B 0,C 180,E1 -11642.322,E2 -11642.322} C_VEL
LIN {X 0,Y 519.406,Z 930.161,A -85,B 0,C 180,E1 -11644.269,E2 -11644.269} C_VEL
LIN {X 0,Y 522.899,Z 911.865,A -85,B 0,C 180,E1 -11645.745,E2 -11645.745} C_VEL
LIN {X 0,Y 527.002,Z 889.186,A -85,B 0,C 180,E1 -11647.315,E2 -11647.315} C_VEL
LIN {X 0,Y 530.13,Z 870.285,A -85,B 0,C 180,E1 -11648.424,E2 -11648.424} C_VEL
LIN {X 0,Y 533.476,Z 848.48,A -85,B 0,C 180,E1 -11649.518,E2 -11649.518} C_VEL
LIN {X 0,Y 536.42,Z 825.839,A -85,B 0,C 180,E1 -11650.442,E2 -11650.442} C_VEL
LIN {X 0,Y 538.743,Z 805.464,A -85,B 0,C 180,E1 -11651.119,E2 -11651.119} C_VEL
LIN {X 0,Y 541.062,Z 780.243,A -85,B 0,C 180,E1 -11651.766,E2 -11651.766} C_VEL
LIN {X 0,Y 542.453,Z 757.686,A -85,B 0,C 180,E1 -11652.185,E2 -11652.185} C_VEL
LIN {X 0,Y 550.682,Z 515.438,A -85,B 0,C 180,E1 -11655.697,E2 -11655.697} C_VEL
LIN {X 0,Y 553.002,Z 446.986,A -85,B 0,C 180,E1 -11656.703,E2 -11656.703} C_VEL
LIN {X 0,Y 541.187,Z 426.742,A -85,B 0,C 180,E1 -11658.431,E2 -11658.431} C_VEL
LIN {X 0,Y 529.583,Z 408.174,A -85,B 0,C 180,E1 -11660.239,E2 -11660.239} C_VEL
LIN {X 0,Y 516.524,Z 388.892,A -85,B 0,C 180,E1 -11662.426,E2 -11662.426} C_VEL
LIN {X 0,Y 507,Z 375.797,A -85,B 0,C 180,E1 -11664.145,E2 -11664.145} C_VEL
LIN {X 0,Y 502.511,Z 369.554,A -85,B 0,C 180,E1 -11665.036,E2 -11665.036} C_VEL
LIN {X 0,Y 501.534,Z 367.315,A -85,B 0,C 180,E1 -11665.514,E2 -11665.514} C_VEL
LIN {X 0,Y 499.515,Z 363.117,A -85,B 0,C 180,E1 -11666.463,E2 -11666.463} C_VEL
LIN {X 0,Y 498.069,Z 359.997,A -85,B 0,C 180,E1 -11667.178,E2 -11667.178} C_VEL
LIN {X 0,Y 497.915,Z 359.205,A -85,B 0,C 180,E1 -11667.368,E2 -11667.368} C_VEL
LIN {X 0,Y 497.891,Z 359.208,A -85,B 0,C 180,E1 -11670.658,E2 -11670.658} C_VEL
LIN {X 0,Y 497.875,Z 359.212,A -85,B 0,C 180,E1 -11674.163,E2 -11674.163} C_VEL
LIN {X 0,Y 497.916,Z 359.207,A -85,B 0,C 180,E1 -11677.57,E2 -11677.57} C_VEL
LIN {X 0,Y 497.907,Z 359.201,A -85,B 0,C 180,E1 -11681.059,E2 -11681.059} C_VEL
LIN {X 0,Y 497.87,Z 359.193,A -85,B 0,C 180,E1 -11684.508,E2 -11684.508} C_VEL
LIN {X 0,Y 497.891,Z 359.186,A -85,B 0,C 180,E1 -11687.964,E2 -11687.964} C_VEL
LIN {X 0,Y 497.927,Z 359.194,A -85,B 0,C 180,E1 -11691.454,E2 -11691.454} C_VEL
LIN {X 0,Y 497.877,Z 359.212,A -85,B 0,C 180,E1 -11694.815,E2 -11694.815} C_VEL
LIN {X 0,Y 497.879,Z 359.195,A -85,B 0,C 180,E1 -11698.389,E2 -11698.389} C_VEL
LIN {X 0,Y 497.927,Z 359.182,A -85,B 0,C 180,E1 -11701.726,E2 -11701.726} C_VEL
LIN {X 0,Y 497.886,Z 359.208,A -85,B 0,C 180,E1 -11705.185,E2 -11705.185} C_VEL
LIN {X 0,Y 497.877,Z 359.213,A -85,B 0,C 180,E1 -11708.663,E2 -11708.663} C_VEL
LIN {X 0,Y 497.921,Z 359.184,A -85,B 0,C 180,E1 -11712.055,E2 -11712.055} C_VEL
LIN {X 0,Y 497.889,Z 359.189,A -85,B 0,C 180,E1 -11715.429,E2 -11715.429} C_VEL
LIN {X 0,Y 497.878,Z 359.203,A -85,B 0,C 180,E1 -11718.931,E2 -11718.931} C_VEL
LIN {X 0,Y 497.911,Z 359.208,A -85,B 0,C 180,E1 -11722.43,E2 -11722.43} C_VEL
LIN {X 0,Y 497.923,Z 359.208,A -85,B 0,C 180,E1 -11725.962,E2 -11725.962} C_VEL
LIN {X 0,Y 497.882,Z 359.212,A -85,B 0,C 180,E1 -11729.356,E2 -11729.356} C_VEL
LIN {X 0,Y 497.886,Z 359.214,A -85,B 0,C 180,E1 -11732.973,E2 -11732.973} C_VEL
LIN {X 0,Y 497.96,Z 359.429,A -85,B 0,C 180,E1 -11734.413,E2 -11734.413} C_VEL
LIN {X 0,Y 499.088,Z 362.488,A -85,B 0,C 180,E1 -11734.679,E2 -11734.679} C_VEL
LIN {X 0,Y 501.677,Z 365.054,A -85,B 0,C 180,E1 -11735.17,E2 -11735.17} C_VEL
LIN {X 0,Y 502.545,Z 365.913,A -85,B 0,C 180,E1 -11735.332,E2 -11735.332} C_VEL
LIN {X 0,Y 504.975,Z 369.615,A -85,B 0,C 180,E1 -11735.811,E2 -11735.811} C_VEL
LIN {X 0,Y 507.1,Z 371.772,A -85,B 0,C 180,E1 -11736.196,E2 -11736.196} C_VEL
LIN {X 0,Y 510.233,Z 375.986,A -85,B 0,C 180,E1 -11736.776,E2 -11736.776} C_VEL
LIN {X 0,Y 512.101,Z 378.284,A -85,B 0,C 180,E1 -11737.109,E2 -11737.109} C_VEL
LIN {X 0,Y 516.665,Z 384.3,A -85,B 0,C 180,E1 -11737.912,E2 -11737.912} C_VEL
LIN {X 0,Y 523.549,Z 393.244,A -85,B 0,C 180,E1 -11739.068,E2 -11739.068} C_VEL
LIN {X 0,Y 535.006,Z 409.148,A -85,B 0,C 180,E1 -11740.889,E2 -11740.889} C_VEL
LIN {X 0,Y 543.992,Z 422.796,A -85,B 0,C 180,E1 -11742.243,E2 -11742.243} C_VEL
LIN {X 0,Y 553.203,Z 438.219,A -85,B 0,C 180,E1 -11743.577,E2 -11743.577} C_VEL
LIN {X 0,Y 544.572,Z 687.444,A -85,B 0,C 180,E1 -11747.186,E2 -11747.186} C_VEL
LIN {X 0,Y 542.48,Z 744.612,A -85,B 0,C 180,E1 -11748.038,E2 -11748.038} C_VEL
LIN {X 0,Y 540.705,Z 769.012,A -85,B 0,C 180,E1 -11748.572,E2 -11748.572} C_VEL
LIN {X 0,Y 538.636,Z 790.891,A -85,B 0,C 180,E1 -11749.206,E2 -11749.206} C_VEL
LIN {X 0,Y 535.917,Z 814.249,A -85,B 0,C 180,E1 -11750.073,E2 -11750.073} C_VEL
LIN {X 0,Y 533.108,Z 834.751,A -85,B 0,C 180,E1 -11751.005,E2 -11751.005} C_VEL
LIN {X 0,Y 529.636,Z 857.24,A -85,B 0,C 180,E1 -11752.221,E2 -11752.221} C_VEL
LIN {X 0,Y 526.195,Z 877.059,A -85,B 0,C 180,E1 -11753.504,E2 -11753.504} C_VEL
LIN {X 0,Y 522.53,Z 896.923,A -85,B 0,C 180,E1 -11754.985,E2 -11754.985} C_VEL
LIN {X 0,Y 519.189,Z 913.758,A -85,B 0,C 180,E1 -11756.442,E2 -11756.442} C_VEL
LIN {X 0,Y 517.09,Z 919.774,A -85,B 0,C 180,E1 -11756.944,E2 -11756.944} C_VEL
LIN {X 0,Y 508.428,Z 935.69,A -85,B 0,C 180,E1 -11758.18,E2 -11758.18} C_VEL
LIN {X 0,Y 506.748,Z 940.366,A -85,B 0,C 180,E1 -11758.669,E2 -11758.669} C_VEL
LIN {X 0,Y 503.486,Z 955.28,A -85,B 0,C 180,E1 -11760.494,E2 -11760.494} C_VEL
LIN {X 0,Y 499.833,Z 972.156,A -85,B 0,C 180,E1 -11762.864,E2 -11762.864} C_VEL
LIN {X 0,Y 497.056,Z 985.339,A -85,B 0,C 180,E1 -11765.011,E2 -11765.011} C_VEL
LIN {X 0,Y 494.347,Z 999.056,A -85,B 0,C 180,E1 -11767.571,E2 -11767.571} C_VEL
LIN {X 0,Y 492.274,Z 1010.293,A -85,B 0,C 180,E1 -11770.048,E2 -11770.048} C_VEL
LIN {X 0,Y 490.644,Z 1020.643,A -85,B 0,C 180,E1 -11772.69,E2 -11772.69} C_VEL
LIN {X 0,Y 489.43,Z 1029.478,A -85,B 0,C 180,E1 -11775.447,E2 -11775.447} C_VEL
LIN {X 0,Y 488.715,Z 1036.164,A -85,B 0,C 180,E1 -11777.955,E2 -11777.955} C_VEL
LIN {X 0,Y 488.219,Z 1042.338,A -85,B 0,C 180,E1 -11780.927,E2 -11780.927} C_VEL
LIN {X 0,Y 488.035,Z 1046.139,A -85,B 0,C 180,E1 -11783.412,E2 -11783.412} C_VEL
LIN {X 0,Y 487.955,Z 1049.071,A -85,B 0,C 180,E1 -11786.24,E2 -11786.24} C_VEL
LIN {X 0,Y 487.936,Z 1050.281,A -85,B 0,C 180,E1 -11788.943,E2 -11788.943} C_VEL
LIN {X 0,Y 487.937,Z 1050.255,A -85,B 0,C 180,E1 -11791.292,E2 -11791.292} C_VEL
LIN {X 0,Y 487.963,Z 1048.864,A -85,B 0,C 180,E1 -11794.113,E2 -11794.113} C_VEL
LIN {X 0,Y 488.032,Z 1046.105,A -85,B 0,C 180,E1 -11796.707,E2 -11796.707} C_VEL
LIN {X 0,Y 488.225,Z 1042.285,A -85,B 0,C 180,E1 -11799.196,E2 -11799.196} C_VEL
LIN {X 0,Y 488.726,Z 1036.095,A -85,B 0,C 180,E1 -11802.165,E2 -11802.165} C_VEL
LIN {X 0,Y 489.442,Z 1029.397,A -85,B 0,C 180,E1 -11804.674,E2 -11804.674} C_VEL
LIN {X 0,Y 490.662,Z 1020.531,A -85,B 0,C 180,E1 -11807.431,E2 -11807.431} C_VEL
LIN {X 0,Y 492.302,Z 1010.161,A -85,B 0,C 180,E1 -11810.075,E2 -11810.075} C_VEL
LIN {X 0,Y 494.534,Z 998.109,A -85,B 0,C 180,E1 -11812.717,E2 -11812.717} C_VEL
LIN {X 0,Y 497.244,Z 984.465,A -85,B 0,C 180,E1 -11815.233,E2 -11815.233} C_VEL
LIN {X 0,Y 500.403,Z 969.632,A -85,B 0,C 180,E1 -11817.618,E2 -11817.618} C_VEL
LIN {X 0,Y 503.753,Z 954.113,A -85,B 0,C 180,E1 -11819.75,E2 -11819.75} C_VEL
LIN {X 0,Y 507.385,Z 937.604,A -85,B 0,C 180,E1 -11821.747,E2 -11821.747} C_VEL
